ABB RAPID module: P101.mod

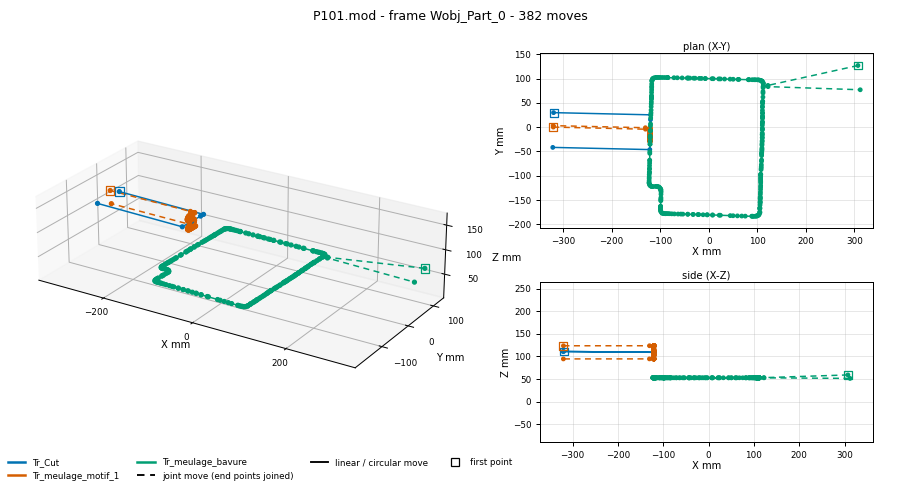
[picture p0: tool path of P101.mod in frame Wobj_Part_0, 382 of 390 moves have a stored position in this frame; points joined in program order, loops and branches not executed]
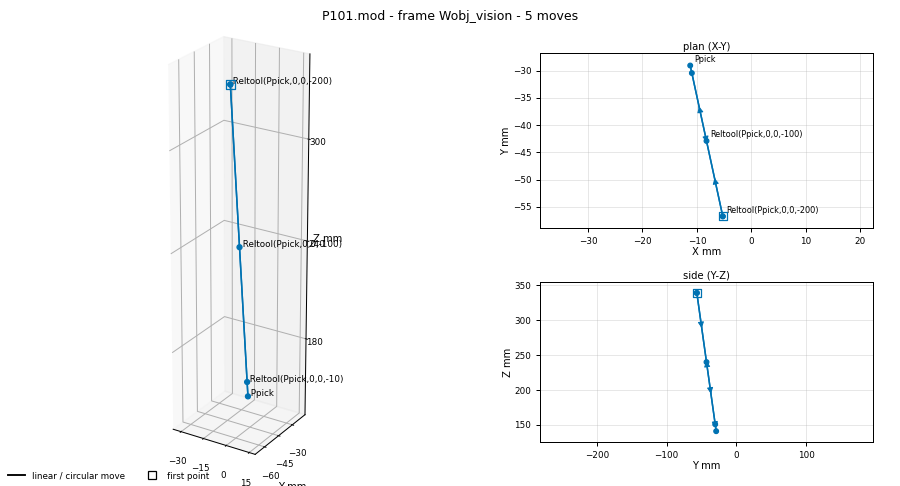
[picture p1: tool path of P101.mod in frame Wobj_vision, 5 of 390 moves have a stored position in this frame; points joined in program order, loops and branches not executed]
MODULE P101
	LOCAL CONST Speeddata vitesse_Tronconnage :=[10, 500, 0, 0];
	LOCAL CONST Robtarget Coupe_0 :=[[-120.682296875,-15.2756298828125,109.2198984375],[0.707017403537071,0.707090697782449,-0.00476918331892896,-0.01124237945003],[0,0,0,0],[8.999999E+09,8.999999E+09,8.999999E+09,8.999999E+09,8.999999E+09,8.999999E+09]];
	LOCAL CONST Robtarget Tr_meulage_motif_1_App1 :=[[-320.249128469475,0.246534065267081,123.638490401036],[0.494425938031671,-0.49422530691975,0.505508072978483,-0.505713284337244],[0,0,0,0],[8.999999E+09,8.999999E+09,8.999999E+09,8.999999E+09,8.999999E+09,8.999999E+09]];
	LOCAL CONST Robtarget Tr_meulage_motif_1_App2 :=[[-130.297538064099,-4.04151394615071,123.715605379427],[0.494425938031671,-0.49422530691975,0.505508072978483,-0.505713284337244],[0,0,0,0],[8.999999E+09,8.999999E+09,8.999999E+09,8.999999E+09,8.999999E+09,8.999999E+09]];
	LOCAL CONST Robtarget Tr_meulage_motif_1_P0 :=[[-120.3000859375,-4.26720068359375,123.7196640625],[0.494425938031671,-0.49422530691975,0.505508072978483,-0.505713284337244],[0,0,0,0],[8.999999E+09,8.999999E+09,8.999999E+09,8.999999E+09,8.999999E+09,8.999999E+09]];
	LOCAL CONST Robtarget Tr_meulage_motif_1_P1 :=[[-120.322734375,-5.2669443359375,123.719625],[0.494425938031671,-0.49422530691975,0.505508072978483,-0.505713284337244],[0,0,0,0],[8.999999E+09,8.999999E+09,8.999999E+09,8.999999E+09,8.999999E+09,8.999999E+09]];
	LOCAL CONST Robtarget Tr_meulage_motif_1_P2 :=[[-120.3453828125,-6.26668798828125,123.71959375],[0.494425938031671,-0.49422530691975,0.505508072978483,-0.505713284337244],[0,0,0,0],[8.999999E+09,8.999999E+09,8.999999E+09,8.999999E+09,8.999999E+09,8.999999E+09]];
	LOCAL CONST Robtarget Tr_meulage_motif_1_P3 :=[[-120.36803125,-7.26643115234375,123.7195625],[0.494425938031671,-0.49422530691975,0.505508072978483,-0.505713284337244],[0,0,0,0],[8.999999E+09,8.999999E+09,8.999999E+09,8.999999E+09,8.999999E+09,8.999999E+09]];
	LOCAL CONST Robtarget Tr_meulage_motif_1_P4 :=[[-120.3906796875,-8.2661748046875,123.7195234375],[0.494425938031671,-0.49422530691975,0.505508072978483,-0.505713284337244],[0,0,0,0],[8.999999E+09,8.999999E+09,8.999999E+09,8.999999E+09,8.999999E+09,8.999999E+09]];
	LOCAL CONST Robtarget Tr_meulage_motif_1_P5 :=[[-120.413328125,-9.26591796875,123.7194921875],[0.494425938031671,-0.49422530691975,0.505508072978483,-0.505713284337244],[0,0,0,0],[8.999999E+09,8.999999E+09,8.999999E+09,8.999999E+09,8.999999E+09,8.999999E+09]];
	LOCAL CONST Robtarget Tr_meulage_motif_1_P6 :=[[-120.4359765625,-10.265662109375,123.7194609375],[0.494425938031671,-0.49422530691975,0.505508072978483,-0.505713284337244],[0,0,0,0],[8.999999E+09,8.999999E+09,8.999999E+09,8.999999E+09,8.999999E+09,8.999999E+09]];
	LOCAL CONST Robtarget Tr_meulage_motif_1_P7 :=[[-120.458625,-11.2654052734375,123.719421875],[0.494425938031671,-0.49422530691975,0.505508072978483,-0.505713284337244],[0,0,0,0],[8.999999E+09,8.999999E+09,8.999999E+09,8.999999E+09,8.999999E+09,8.999999E+09]];
	LOCAL CONST Robtarget Tr_meulage_motif_1_P8 :=[[-120.481265625,-12.2651484375,123.719390625],[0.494425938031671,-0.49422530691975,0.505508072978483,-0.505713284337244],[0,0,0,0],[8.999999E+09,8.999999E+09,8.999999E+09,8.999999E+09,8.999999E+09,8.999999E+09]];
	LOCAL CONST Robtarget Tr_meulage_motif_1_P9 :=[[-120.5039140625,-13.264892578125,123.719359375],[0.494425938031671,-0.49422530691975,0.505508072978483,-0.505713284337244],[0,0,0,0],[8.999999E+09,8.999999E+09,8.999999E+09,8.999999E+09,8.999999E+09,8.999999E+09]];
	LOCAL CONST Robtarget Tr_meulage_motif_1_P10 :=[[-120.5265625,-14.2646357421875,123.719328125],[0.494425938031671,-0.49422530691975,0.505508072978483,-0.505713284337244],[0,0,0,0],[8.999999E+09,8.999999E+09,8.999999E+09,8.999999E+09,8.999999E+09,8.999999E+09]];
	LOCAL CONST Robtarget Tr_meulage_motif_1_P11 :=[[-120.5492109375,-15.26437890625,123.7192890625],[0.494425938031671,-0.49422530691975,0.505508072978483,-0.505713284337244],[0,0,0,0],[8.999999E+09,8.999999E+09,8.999999E+09,8.999999E+09,8.999999E+09,8.999999E+09]];
	LOCAL CONST Robtarget Tr_meulage_motif_1_P12 :=[[-120.571859375,-16.264123046875,123.7192578125],[0.494425938031671,-0.49422530691975,0.505508072978483,-0.505713284337244],[0,0,0,0],[8.999999E+09,8.999999E+09,8.999999E+09,8.999999E+09,8.999999E+09,8.999999E+09]];
	LOCAL CONST Robtarget Tr_meulage_motif_1_P13 :=[[-120.5945078125,-17.2638671875,123.7192265625],[0.494425938031671,-0.49422530691975,0.505508072978483,-0.505713284337244],[0,0,0,0],[8.999999E+09,8.999999E+09,8.999999E+09,8.999999E+09,8.999999E+09,8.999999E+09]];
	LOCAL CONST Robtarget Tr_meulage_motif_1_P14 :=[[-120.61715625,-18.263609375,123.7191875],[0.494425938031671,-0.49422530691975,0.505508072978483,-0.505713284337244],[0,0,0,0],[8.999999E+09,8.999999E+09,8.999999E+09,8.999999E+09,8.999999E+09,8.999999E+09]];
	LOCAL CONST Robtarget Tr_meulage_motif_1_P15 :=[[-120.6398046875,-19.263353515625,123.71915625],[0.494425938031671,-0.49422530691975,0.505508072978483,-0.505713284337244],[0,0,0,0],[8.999999E+09,8.999999E+09,8.999999E+09,8.999999E+09,8.999999E+09,8.999999E+09]];
	LOCAL CONST Robtarget Tr_meulage_motif_1_P16 :=[[-120.662453125,-20.26309765625,123.719125],[0.494425938031671,-0.49422530691975,0.505508072978483,-0.505713284337244],[0,0,0,0],[8.999999E+09,8.999999E+09,8.999999E+09,8.999999E+09,8.999999E+09,8.999999E+09]];
	LOCAL CONST Robtarget Tr_meulage_motif_1_P17 :=[[-120.6851015625,-21.26283984375,123.7190859375],[0.494425938031671,-0.49422530691975,0.505508072978483,-0.505713284337244],[0,0,0,0],[8.999999E+09,8.999999E+09,8.999999E+09,8.999999E+09,8.999999E+09,8.999999E+09]];
	LOCAL CONST Robtarget Tr_meulage_motif_1_P18 :=[[-120.70775,-22.262583984375,123.7190546875],[0.494425938031671,-0.49422530691975,0.505508072978483,-0.505713284337244],[0,0,0,0],[8.999999E+09,8.999999E+09,8.999999E+09,8.999999E+09,8.999999E+09,8.999999E+09]];
	LOCAL CONST Robtarget Tr_meulage_motif_1_P19 :=[[-120.7312421875,-23.254865234375,123.6084296875],[0.494425938031671,-0.49422530691975,0.505508072978483,-0.505713284337244],[0,0,0,0],[8.999999E+09,8.999999E+09,8.999999E+09,8.999999E+09,8.999999E+09,8.999999E+09]];
	LOCAL CONST Robtarget Tr_meulage_motif_1_P20 :=[[-120.754609375,-24.201072265625,123.39721875],[0.494425938031671,-0.49422530691975,0.505508072978483,-0.505713284337244],[0,0,0,0],[8.999999E+09,8.999999E+09,8.999999E+09,8.999999E+09,8.999999E+09,8.999999E+09]];
	LOCAL CONST Robtarget Tr_meulage_motif_1_P21 :=[[-120.7764140625,-25.053505859375,123.125359375],[0.494425938031671,-0.49422530691975,0.505508072978483,-0.505713284337244],[0,0,0,0],[8.999999E+09,8.999999E+09,8.999999E+09,8.999999E+09,8.999999E+09,8.999999E+09]];
	LOCAL CONST Robtarget Tr_meulage_motif_1_P22 :=[[-120.795921875,-25.80318359375,122.84940625],[0.494425938031671,-0.49422530691975,0.505508072978483,-0.505713284337244],[0,0,0,0],[8.999999E+09,8.999999E+09,8.999999E+09,8.999999E+09,8.999999E+09,8.999999E+09]];
	LOCAL CONST Robtarget Tr_meulage_motif_1_P23 :=[[-120.8265,-26.90381640625,122.2332734375],[0.494425938031671,-0.49422530691975,0.505508072978483,-0.505713284337244],[0,0,0,0],[8.999999E+09,8.999999E+09,8.999999E+09,8.999999E+09,8.999999E+09,8.999999E+09]];
	LOCAL CONST Robtarget Tr_meulage_motif_1_P24 :=[[-120.8574453125,-27.927224609375,121.3856171875],[0.494425938031671,-0.49422530691975,0.505508072978483,-0.505713284337244],[0,0,0,0],[8.999999E+09,8.999999E+09,8.999999E+09,8.999999E+09,8.999999E+09,8.999999E+09]];
	LOCAL CONST Robtarget Tr_meulage_motif_1_P25 :=[[-120.8860234375,-28.774416015625,120.3617578125],[0.494425938031671,-0.49422530691975,0.505508072978483,-0.505713284337244],[0,0,0,0],[8.999999E+09,8.999999E+09,8.999999E+09,8.999999E+09,8.999999E+09,8.999999E+09]];
	LOCAL CONST Robtarget Tr_meulage_motif_1_P26 :=[[-120.907296875,-29.262177734375,119.2456015625],[0.494425938031671,-0.49422530691975,0.505508072978483,-0.505713284337244],[0,0,0,0],[8.999999E+09,8.999999E+09,8.999999E+09,8.999999E+09,8.999999E+09,8.999999E+09]];
	LOCAL CONST Robtarget Tr_meulage_motif_1_P27 :=[[-120.91428125,-29.28906640625,118.5496640625],[0.494425938031671,-0.49422530691975,0.505508072978483,-0.505713284337244],[0,0,0,0],[8.999999E+09,8.999999E+09,8.999999E+09,8.999999E+09,8.999999E+09,8.999999E+09]];
	LOCAL CONST Robtarget Tr_meulage_motif_1_P28 :=[[-120.9203359375,-29.28890625,117.8884375],[0.494425938031671,-0.49422530691975,0.505508072978483,-0.505713284337244],[0,0,0,0],[8.999999E+09,8.999999E+09,8.999999E+09,8.999999E+09,8.999999E+09,8.999999E+09]];
	LOCAL CONST Robtarget Tr_meulage_motif_1_P29 :=[[-120.925140625,-29.23388671875,117.227375],[0.494425938031671,-0.49422530691975,0.505508072978483,-0.505713284337244],[0,0,0,0],[8.999999E+09,8.999999E+09,8.999999E+09,8.999999E+09,8.999999E+09,8.999999E+09]];
	LOCAL CONST Robtarget Tr_meulage_motif_1_P30 :=[[-120.9239453125,-28.735529296875,116.1256875],[0.494425938031671,-0.49422530691975,0.505508072978483,-0.505713284337244],[0,0,0,0],[8.999999E+09,8.999999E+09,8.999999E+09,8.999999E+09,8.999999E+09,8.999999E+09]];
	LOCAL CONST Robtarget Tr_meulage_motif_1_P31 :=[[-120.9137578125,-27.878880859375,115.1191328125],[0.494425938031671,-0.49422530691975,0.505508072978483,-0.505713284337244],[0,0,0,0],[8.999999E+09,8.999999E+09,8.999999E+09,8.999999E+09,8.999999E+09,8.999999E+09]];
	LOCAL CONST Robtarget Tr_meulage_motif_1_P32 :=[[-120.898171875,-26.855537109375,114.290328125],[0.494425938031671,-0.49422530691975,0.505508072978483,-0.505713284337244],[0,0,0,0],[8.999999E+09,8.999999E+09,8.999999E+09,8.999999E+09,8.999999E+09,8.999999E+09]];
	LOCAL CONST Robtarget Tr_meulage_motif_1_P33 :=[[-120.886234375,-26.168525390625,113.8946171875],[0.494425938031671,-0.49422530691975,0.505508072978483,-0.505713284337244],[0,0,0,0],[8.999999E+09,8.999999E+09,8.999999E+09,8.999999E+09,8.999999E+09,8.999999E+09]];
	LOCAL CONST Robtarget Tr_meulage_motif_1_P34 :=[[-120.86446875,-25.010548828125,113.4071484375],[0.494425938031671,-0.49422530691975,0.505508072978483,-0.505713284337244],[0,0,0,0],[8.999999E+09,8.999999E+09,8.999999E+09,8.999999E+09,8.999999E+09,8.999999E+09]];
	LOCAL CONST Robtarget Tr_meulage_motif_1_P35 :=[[-120.8477421875,-24.165669921875,113.14309375],[0.494425938031671,-0.49422530691975,0.505508072978483,-0.505713284337244],[0,0,0,0],[8.999999E+09,8.999999E+09,8.999999E+09,8.999999E+09,8.999999E+09,8.999999E+09]];
	LOCAL CONST Robtarget Tr_meulage_motif_1_P36 :=[[-120.8285078125,-23.233859375,112.9386640625],[0.494425938031671,-0.49422530691975,0.505508072978483,-0.505713284337244],[0,0,0,0],[8.999999E+09,8.999999E+09,8.999999E+09,8.999999E+09,8.999999E+09,8.999999E+09]];
	LOCAL CONST Robtarget Tr_meulage_motif_1_P37 :=[[-120.8072734375,-22.2525234375,112.830109375],[0.494425938031671,-0.49422530691975,0.505508072978483,-0.505713284337244],[0,0,0,0],[8.999999E+09,8.999999E+09,8.999999E+09,8.999999E+09,8.999999E+09,8.999999E+09]];
	LOCAL CONST Robtarget Tr_meulage_motif_1_P38 :=[[-120.7858046875,-21.2601875,112.719546875],[0.494425938031671,-0.49422530691975,0.505508072978483,-0.505713284337244],[0,0,0,0],[8.999999E+09,8.999999E+09,8.999999E+09,8.999999E+09,8.999999E+09,8.999999E+09]];
	LOCAL CONST Robtarget Tr_meulage_motif_1_P39 :=[[-120.76315625,-20.2604453125,112.7195859375],[0.494425938031671,-0.49422530691975,0.505508072978483,-0.505713284337244],[0,0,0,0],[8.999999E+09,8.999999E+09,8.999999E+09,8.999999E+09,8.999999E+09,8.999999E+09]];
	LOCAL CONST Robtarget Tr_meulage_motif_1_P40 :=[[-120.7405078125,-19.260701171875,112.7196171875],[0.494425938031671,-0.49422530691975,0.505508072978483,-0.505713284337244],[0,0,0,0],[8.999999E+09,8.999999E+09,8.999999E+09,8.999999E+09,8.999999E+09,8.999999E+09]];
	LOCAL CONST Robtarget Tr_meulage_motif_1_P41 :=[[-120.7178671875,-18.26095703125,112.7196484375],[0.494425938031671,-0.49422530691975,0.505508072978483,-0.505713284337244],[0,0,0,0],[8.999999E+09,8.999999E+09,8.999999E+09,8.999999E+09,8.999999E+09,8.999999E+09]];
	LOCAL CONST Robtarget Tr_meulage_motif_1_P42 :=[[-120.69521875,-17.26121484375,112.7196875],[0.494425938031671,-0.49422530691975,0.505508072978483,-0.505713284337244],[0,0,0,0],[8.999999E+09,8.999999E+09,8.999999E+09,8.999999E+09,8.999999E+09,8.999999E+09]];
	LOCAL CONST Robtarget Tr_meulage_motif_1_P43 :=[[-120.6725703125,-16.261470703125,112.71971875],[0.494425938031671,-0.49422530691975,0.505508072978483,-0.505713284337244],[0,0,0,0],[8.999999E+09,8.999999E+09,8.999999E+09,8.999999E+09,8.999999E+09,8.999999E+09]];
	LOCAL CONST Robtarget Tr_meulage_motif_1_P44 :=[[-120.649921875,-15.2617275390625,112.71975],[0.494425938031671,-0.49422530691975,0.505508072978483,-0.505713284337244],[0,0,0,0],[8.999999E+09,8.999999E+09,8.999999E+09,8.999999E+09,8.999999E+09,8.999999E+09]];
	LOCAL CONST Robtarget Tr_meulage_motif_1_P45 :=[[-120.6272734375,-14.261984375,112.7197890625],[0.494425938031671,-0.49422530691975,0.505508072978483,-0.505713284337244],[0,0,0,0],[8.999999E+09,8.999999E+09,8.999999E+09,8.999999E+09,8.999999E+09,8.999999E+09]];
	LOCAL CONST Robtarget Tr_meulage_motif_1_P46 :=[[-120.604625,-13.262240234375,112.7198203125],[0.494425938031671,-0.49422530691975,0.505508072978483,-0.505713284337244],[0,0,0,0],[8.999999E+09,8.999999E+09,8.999999E+09,8.999999E+09,8.999999E+09,8.999999E+09]];
	LOCAL CONST Robtarget Tr_meulage_motif_1_P47 :=[[-120.5819765625,-12.2624970703125,112.7198515625],[0.494425938031671,-0.49422530691975,0.505508072978483,-0.505713284337244],[0,0,0,0],[8.999999E+09,8.999999E+09,8.999999E+09,8.999999E+09,8.999999E+09,8.999999E+09]];
	LOCAL CONST Robtarget Tr_meulage_motif_1_P48 :=[[-120.559328125,-11.26275390625,112.719890625],[0.494425938031671,-0.49422530691975,0.505508072978483,-0.505713284337244],[0,0,0,0],[8.999999E+09,8.999999E+09,8.999999E+09,8.999999E+09,8.999999E+09,8.999999E+09]];
	LOCAL CONST Robtarget Tr_meulage_motif_1_P49 :=[[-120.537859375,-10.2704189453125,112.609328125],[0.494425938031671,-0.49422530691975,0.505508072978483,-0.505713284337244],[0,0,0,0],[8.999999E+09,8.999999E+09,8.999999E+09,8.999999E+09,8.999999E+09,8.999999E+09]];
	LOCAL CONST Robtarget Tr_meulage_motif_1_P50 :=[[-120.518359375,-9.3241103515625,112.3981875],[0.494425938031671,-0.49422530691975,0.505508072978483,-0.505713284337244],[0,0,0,0],[8.999999E+09,8.999999E+09,8.999999E+09,8.999999E+09,8.999999E+09,8.999999E+09]];
	LOCAL CONST Robtarget Tr_meulage_motif_1_P51 :=[[-120.50153125,-8.471544921875,112.1263828125],[0.494425938031671,-0.49422530691975,0.505508072978483,-0.505713284337244],[0,0,0,0],[8.999999E+09,8.999999E+09,8.999999E+09,8.999999E+09,8.999999E+09,8.999999E+09]];
	LOCAL CONST Robtarget Tr_meulage_motif_1_P52 :=[[-120.488203125,-7.760154296875,111.8222578125],[0.494425938031671,-0.49422530691975,0.505508072978483,-0.505713284337244],[0,0,0,0],[8.999999E+09,8.999999E+09,8.999999E+09,8.999999E+09,8.999999E+09,8.999999E+09]];
	LOCAL CONST Robtarget Tr_meulage_motif_1_P53 :=[[-120.47084375,-6.725791015625,111.1597890625],[0.494425938031671,-0.49422530691975,0.505508072978483,-0.505713284337244],[0,0,0,0],[8.999999E+09,8.999999E+09,8.999999E+09,8.999999E+09,8.999999E+09,8.999999E+09]];
	LOCAL CONST Robtarget Tr_meulage_motif_1_P54 :=[[-120.458671875,-5.82386767578125,110.257921875],[0.494425938031671,-0.49422530691975,0.505508072978483,-0.505713284337244],[0,0,0,0],[8.999999E+09,8.999999E+09,8.999999E+09,8.999999E+09,8.999999E+09,8.999999E+09]];
	LOCAL CONST Robtarget Tr_meulage_motif_1_P55 :=[[-120.4561328125,-5.28878369140625,109.211953125],[0.494425938031671,-0.49422530691975,0.505508072978483,-0.505713284337244],[0,0,0,0],[8.999999E+09,8.999999E+09,8.999999E+09,8.999999E+09,8.999999E+09,8.999999E+09]];
	LOCAL CONST Robtarget Tr_meulage_motif_1_P56 :=[[-120.458296875,-5.1038828125,108.5187734375],[0.494425938031671,-0.49422530691975,0.505508072978483,-0.505713284337244],[0,0,0,0],[8.999999E+09,8.999999E+09,8.999999E+09,8.999999E+09,8.999999E+09,8.999999E+09]];
	LOCAL CONST Robtarget Tr_meulage_motif_1_P57 :=[[-120.4638984375,-5.0398701171875,107.7488046875],[0.494425938031671,-0.49422530691975,0.505508072978483,-0.505713284337244],[0,0,0,0],[8.999999E+09,8.999999E+09,8.999999E+09,8.999999E+09,8.999999E+09,8.999999E+09]];
	LOCAL CONST Robtarget Tr_meulage_motif_1_P58 :=[[-120.4724609375,-5.1066044921875,106.9789609375],[0.494425938031671,-0.49422530691975,0.505508072978483,-0.505713284337244],[0,0,0,0],[8.999999E+09,8.999999E+09,8.999999E+09,8.999999E+09,8.999999E+09,8.999999E+09]];
	LOCAL CONST Robtarget Tr_meulage_motif_1_P59 :=[[-120.492109375,-5.52582373046875,105.8707421875],[0.494425938031671,-0.49422530691975,0.505508072978483,-0.505713284337244],[0,0,0,0],[8.999999E+09,8.999999E+09,8.999999E+09,8.999999E+09,8.999999E+09,8.999999E+09]];
	LOCAL CONST Robtarget Tr_meulage_motif_1_P60 :=[[-120.506859375,-5.939888671875,105.2850625],[0.494425938031671,-0.49422530691975,0.505508072978483,-0.505713284337244],[0,0,0,0],[8.999999E+09,8.999999E+09,8.999999E+09,8.999999E+09,8.999999E+09,8.999999E+09]];
	LOCAL CONST Robtarget Tr_meulage_motif_1_P61 :=[[-120.5350703125,-6.826572265625,104.3979453125],[0.494425938031671,-0.49422530691975,0.505508072978483,-0.505713284337244],[0,0,0,0],[8.999999E+09,8.999999E+09,8.999999E+09,8.999999E+09,8.999999E+09,8.999999E+09]];
	LOCAL CONST Robtarget Tr_meulage_motif_1_P62 :=[[-120.552125,-7.412009765625,103.9836328125],[0.494425938031671,-0.49422530691975,0.505508072978483,-0.505713284337244],[0,0,0,0],[8.999999E+09,8.999999E+09,8.999999E+09,8.999999E+09,8.999999E+09,8.999999E+09]];
	LOCAL CONST Robtarget Tr_meulage_motif_1_P63 :=[[-120.5824296875,-8.529498046875,103.4395234375],[0.494425938031671,-0.49422530691975,0.505508072978483,-0.505713284337244],[0,0,0,0],[8.999999E+09,8.999999E+09,8.999999E+09,8.999999E+09,8.999999E+09,8.999999E+09]];
	LOCAL CONST Robtarget Tr_meulage_motif_1_P64 :=[[-120.603828125,-9.35480859375,103.1440078125],[0.494425938031671,-0.49422530691975,0.505508072978483,-0.505713284337244],[0,0,0,0],[8.999999E+09,8.999999E+09,8.999999E+09,8.999999E+09,8.999999E+09,8.999999E+09]];
	LOCAL CONST Robtarget Tr_meulage_motif_1_P65 :=[[-120.6268125,-10.2865205078125,102.939515625],[0.494425938031671,-0.49422530691975,0.505508072978483,-0.505713284337244],[0,0,0,0],[8.999999E+09,8.999999E+09,8.999999E+09,8.999999E+09,8.999999E+09,8.999999E+09]];
	LOCAL CONST Robtarget Tr_meulage_motif_1_P66 :=[[-120.6500390625,-11.2678046875,102.8308984375],[0.494425938031671,-0.49422530691975,0.505508072978483,-0.505713284337244],[0,0,0,0],[8.999999E+09,8.999999E+09,8.999999E+09,8.999999E+09,8.999999E+09,8.999999E+09]];
	LOCAL CONST Robtarget Tr_meulage_motif_1_P67 :=[[-120.67353125,-12.2600859375,102.7202734375],[0.494425938031671,-0.49422530691975,0.505508072978483,-0.505713284337244],[0,0,0,0],[8.999999E+09,8.999999E+09,8.999999E+09,8.999999E+09,8.999999E+09,8.999999E+09]];
	LOCAL CONST Robtarget Tr_meulage_motif_1_P68 :=[[-120.696171875,-13.259830078125,102.7202421875],[0.494425938031671,-0.49422530691975,0.505508072978483,-0.505713284337244],[0,0,0,0],[8.999999E+09,8.999999E+09,8.999999E+09,8.999999E+09,8.999999E+09,8.999999E+09]];
	LOCAL CONST Robtarget Tr_meulage_motif_1_P69 :=[[-120.7188203125,-14.2595732421875,102.720203125],[0.494425938031671,-0.49422530691975,0.505508072978483,-0.505713284337244],[0,0,0,0],[8.999999E+09,8.999999E+09,8.999999E+09,8.999999E+09,8.999999E+09,8.999999E+09]];
	LOCAL CONST Robtarget Tr_meulage_motif_1_P70 :=[[-120.74146875,-15.25931640625,102.720171875],[0.494425938031671,-0.49422530691975,0.505508072978483,-0.505713284337244],[0,0,0,0],[8.999999E+09,8.999999E+09,8.999999E+09,8.999999E+09,8.999999E+09,8.999999E+09]];
	LOCAL CONST Robtarget Tr_meulage_motif_1_P71 :=[[-120.7641171875,-16.259060546875,102.720140625],[0.494425938031671,-0.49422530691975,0.505508072978483,-0.505713284337244],[0,0,0,0],[8.999999E+09,8.999999E+09,8.999999E+09,8.999999E+09,8.999999E+09,8.999999E+09]];
	LOCAL CONST Robtarget Tr_meulage_motif_1_P72 :=[[-120.786765625,-17.258802734375,102.7201015625],[0.494425938031671,-0.49422530691975,0.505508072978483,-0.505713284337244],[0,0,0,0],[8.999999E+09,8.999999E+09,8.999999E+09,8.999999E+09,8.999999E+09,8.999999E+09]];
	LOCAL CONST Robtarget Tr_meulage_motif_1_P73 :=[[-120.8094140625,-18.258546875,102.7200703125],[0.494425938031671,-0.49422530691975,0.505508072978483,-0.505713284337244],[0,0,0,0],[8.999999E+09,8.999999E+09,8.999999E+09,8.999999E+09,8.999999E+09,8.999999E+09]];
	LOCAL CONST Robtarget Tr_meulage_motif_1_P74 :=[[-120.8320625,-19.258291015625,102.7200390625],[0.494425938031671,-0.49422530691975,0.505508072978483,-0.505713284337244],[0,0,0,0],[8.999999E+09,8.999999E+09,8.999999E+09,8.999999E+09,8.999999E+09,8.999999E+09]];
	LOCAL CONST Robtarget Tr_meulage_motif_1_P75 :=[[-120.8547109375,-20.258033203125,102.72],[0.494425938031671,-0.49422530691975,0.505508072978483,-0.505713284337244],[0,0,0,0],[8.999999E+09,8.999999E+09,8.999999E+09,8.999999E+09,8.999999E+09,8.999999E+09]];
	LOCAL CONST Robtarget Tr_meulage_motif_1_P76 :=[[-120.877359375,-21.25777734375,102.71996875],[0.494425938031671,-0.49422530691975,0.505508072978483,-0.505713284337244],[0,0,0,0],[8.999999E+09,8.999999E+09,8.999999E+09,8.999999E+09,8.999999E+09,8.999999E+09]];
	LOCAL CONST Robtarget Tr_meulage_motif_1_P77 :=[[-120.9000078125,-22.257521484375,102.7199375],[0.494425938031671,-0.49422530691975,0.505508072978483,-0.505713284337244],[0,0,0,0],[8.999999E+09,8.999999E+09,8.999999E+09,8.999999E+09,8.999999E+09,8.999999E+09]];
	LOCAL CONST Robtarget Tr_meulage_motif_1_P78 :=[[-120.9235,-23.249802734375,102.6093125],[0.494425938031671,-0.49422530691975,0.505508072978483,-0.505713284337244],[0,0,0,0],[8.999999E+09,8.999999E+09,8.999999E+09,8.999999E+09,8.999999E+09,8.999999E+09]];
	LOCAL CONST Robtarget Tr_meulage_motif_1_P79 :=[[-120.9468671875,-24.1960078125,102.3981015625],[0.494425938031671,-0.49422530691975,0.505508072978483,-0.505713284337244],[0,0,0,0],[8.999999E+09,8.999999E+09,8.999999E+09,8.999999E+09,8.999999E+09,8.999999E+09]];
	LOCAL CONST Robtarget Tr_meulage_motif_1_P80 :=[[-120.968671875,-25.048443359375,102.1262421875],[0.494425938031671,-0.49422530691975,0.505508072978483,-0.505713284337244],[0,0,0,0],[8.999999E+09,8.999999E+09,8.999999E+09,8.999999E+09,8.999999E+09,8.999999E+09]];
	LOCAL CONST Robtarget Tr_meulage_motif_1_P81 :=[[-120.9881796875,-25.79812109375,101.8502890625],[0.494425938031671,-0.49422530691975,0.505508072978483,-0.505713284337244],[0,0,0,0],[8.999999E+09,8.999999E+09,8.999999E+09,8.999999E+09,8.999999E+09,8.999999E+09]];
	LOCAL CONST Robtarget Tr_meulage_motif_1_P82 :=[[-121.0187578125,-26.89875390625,101.23415625],[0.494425938031671,-0.49422530691975,0.505508072978483,-0.505713284337244],[0,0,0,0],[8.999999E+09,8.999999E+09,8.999999E+09,8.999999E+09,8.999999E+09,8.999999E+09]];
	LOCAL CONST Robtarget Tr_meulage_motif_1_P83 :=[[-121.048609375,-27.85501171875,100.3401875],[0.494425938031671,-0.49422530691975,0.505508072978483,-0.505713284337244],[0,0,0,0],[8.999999E+09,8.999999E+09,8.999999E+09,8.999999E+09,8.999999E+09,8.999999E+09]];
	LOCAL CONST Robtarget Tr_meulage_motif_1_P84 :=[[-121.07234375,-28.46371875,99.25421875],[0.494425938031671,-0.49422530691975,0.505508072978483,-0.505713284337244],[0,0,0,0],[8.999999E+09,8.999999E+09,8.999999E+09,8.999999E+09,8.999999E+09,8.999999E+09]];
	LOCAL CONST Robtarget Tr_meulage_motif_1_P85 :=[[-121.0851953125,-28.63275,98.269875],[0.494425938031671,-0.49422530691975,0.505508072978483,-0.505713284337244],[0,0,0,0],[8.999999E+09,8.999999E+09,8.999999E+09,8.999999E+09,8.999999E+09,8.999999E+09]];
	LOCAL CONST Robtarget Tr_meulage_motif_1_P86 :=[[-121.08409375,-28.501265625,98.065234375],[0.494425938031671,-0.49422530691975,0.505508072978483,-0.505713284337244],[0,0,0,0],[8.999999E+09,8.999999E+09,8.999999E+09,8.999999E+09,8.999999E+09,8.999999E+09]];
	LOCAL CONST Robtarget Tr_meulage_motif_1_P87 :=[[-121.0879453125,-28.377748046875,97.338859375],[0.494425938031671,-0.49422530691975,0.505508072978483,-0.505713284337244],[0,0,0,0],[8.999999E+09,8.999999E+09,8.999999E+09,8.999999E+09,8.999999E+09,8.999999E+09]];
	LOCAL CONST Robtarget Tr_meulage_motif_1_P88 :=[[-121.08103125,-27.693697265625,96.402015625],[0.494425938031671,-0.49422530691975,0.505508072978483,-0.505713284337244],[0,0,0,0],[8.999999E+09,8.999999E+09,8.999999E+09,8.999999E+09,8.999999E+09,8.999999E+09]];
	LOCAL CONST Robtarget Tr_meulage_motif_1_P89 :=[[-121.0726484375,-27.136103515625,95.9382421875],[0.494425938031671,-0.49422530691975,0.505508072978483,-0.505713284337244],[0,0,0,0],[8.999999E+09,8.999999E+09,8.999999E+09,8.999999E+09,8.999999E+09,8.999999E+09]];
	LOCAL CONST Robtarget Tr_meulage_motif_1_P90 :=[[-121.05190625,-26.005953125,95.4078671875],[0.494425938031671,-0.49422530691975,0.505508072978483,-0.505713284337244],[0,0,0,0],[8.999999E+09,8.999999E+09,8.999999E+09,8.999999E+09,8.999999E+09,8.999999E+09]];
	LOCAL CONST Robtarget Tr_meulage_motif_1_P91 :=[[-121.0351875,-25.16107421875,95.1438125],[0.494425938031671,-0.49422530691975,0.505508072978483,-0.505713284337244],[0,0,0,0],[8.999999E+09,8.999999E+09,8.999999E+09,8.999999E+09,8.999999E+09,8.999999E+09]];
	LOCAL CONST Robtarget Tr_meulage_motif_1_P92 :=[[-121.015953125,-24.229263671875,94.9393828125],[0.494425938031671,-0.49422530691975,0.505508072978483,-0.505713284337244],[0,0,0,0],[8.999999E+09,8.999999E+09,8.999999E+09,8.999999E+09,8.999999E+09,8.999999E+09]];
	LOCAL CONST Robtarget Tr_meulage_motif_1_P93 :=[[-120.99471875,-23.247927734375,94.830828125],[0.494425938031671,-0.49422530691975,0.505508072978483,-0.505713284337244],[0,0,0,0],[8.999999E+09,8.999999E+09,8.999999E+09,8.999999E+09,8.999999E+09,8.999999E+09]];
	LOCAL CONST Robtarget Tr_meulage_motif_1_P94 :=[[-120.97325,-22.255591796875,94.7202734375],[0.494425938031671,-0.49422530691975,0.505508072978483,-0.505713284337244],[0,0,0,0],[8.999999E+09,8.999999E+09,8.999999E+09,8.999999E+09,8.999999E+09,8.999999E+09]];
	LOCAL CONST Robtarget Tr_meulage_motif_1_P95 :=[[-120.9506015625,-21.255849609375,94.7203046875],[0.494425938031671,-0.49422530691975,0.505508072978483,-0.505713284337244],[0,0,0,0],[8.999999E+09,8.999999E+09,8.999999E+09,8.999999E+09,8.999999E+09,8.999999E+09]];
	LOCAL CONST Robtarget Tr_meulage_motif_1_P96 :=[[-120.927953125,-20.25610546875,94.7203359375],[0.494425938031671,-0.49422530691975,0.505508072978483,-0.505713284337244],[0,0,0,0],[8.999999E+09,8.999999E+09,8.999999E+09,8.999999E+09,8.999999E+09,8.999999E+09]];
	LOCAL CONST Robtarget Tr_meulage_motif_1_P97 :=[[-120.9053046875,-19.256361328125,94.720375],[0.494425938031671,-0.49422530691975,0.505508072978483,-0.505713284337244],[0,0,0,0],[8.999999E+09,8.999999E+09,8.999999E+09,8.999999E+09,8.999999E+09,8.999999E+09]];
	LOCAL CONST Robtarget Tr_meulage_motif_1_P98 :=[[-120.88265625,-18.256619140625,94.72040625],[0.494425938031671,-0.49422530691975,0.505508072978483,-0.505713284337244],[0,0,0,0],[8.999999E+09,8.999999E+09,8.999999E+09,8.999999E+09,8.999999E+09,8.999999E+09]];
	LOCAL CONST Robtarget Tr_meulage_motif_1_P99 :=[[-120.8600078125,-17.256875,94.7204375],[0.494425938031671,-0.49422530691975,0.505508072978483,-0.505713284337244],[0,0,0,0],[8.999999E+09,8.999999E+09,8.999999E+09,8.999999E+09,8.999999E+09,8.999999E+09]];
	LOCAL CONST Robtarget Tr_meulage_motif_1_P100 :=[[-120.837359375,-16.2571318359375,94.7204765625],[0.494425938031671,-0.49422530691975,0.505508072978483,-0.505713284337244],[0,0,0,0],[8.999999E+09,8.999999E+09,8.999999E+09,8.999999E+09,8.999999E+09,8.999999E+09]];
	LOCAL CONST Robtarget Tr_meulage_motif_1_P101 :=[[-120.8147109375,-15.2573876953125,94.7205078125],[0.494425938031671,-0.49422530691975,0.505508072978483,-0.505713284337244],[0,0,0,0],[8.999999E+09,8.999999E+09,8.999999E+09,8.999999E+09,8.999999E+09,8.999999E+09]];
	LOCAL CONST Robtarget Tr_meulage_motif_1_P102 :=[[-120.7920625,-14.25764453125,94.7205390625],[0.494425938031671,-0.49422530691975,0.505508072978483,-0.505713284337244],[0,0,0,0],[8.999999E+09,8.999999E+09,8.999999E+09,8.999999E+09,8.999999E+09,8.999999E+09]];
	LOCAL CONST Robtarget Tr_meulage_motif_1_P103 :=[[-120.7694140625,-13.2579013671875,94.720578125],[0.494425938031671,-0.49422530691975,0.505508072978483,-0.505713284337244],[0,0,0,0],[8.999999E+09,8.999999E+09,8.999999E+09,8.999999E+09,8.999999E+09,8.999999E+09]];
	LOCAL CONST Robtarget Tr_meulage_motif_1_P104 :=[[-120.746765625,-12.2581572265625,94.720609375],[0.494425938031671,-0.49422530691975,0.505508072978483,-0.505713284337244],[0,0,0,0],[8.999999E+09,8.999999E+09,8.999999E+09,8.999999E+09,8.999999E+09,8.999999E+09]];
	LOCAL CONST Robtarget Tr_meulage_motif_1_P105 :=[[-120.724125,-11.2584140625,94.720640625],[0.494425938031671,-0.49422530691975,0.505508072978483,-0.505713284337244],[0,0,0,0],[8.999999E+09,8.999999E+09,8.999999E+09,8.999999E+09,8.999999E+09,8.999999E+09]];
	LOCAL CONST Robtarget Tr_meulage_motif_1_P106 :=[[-120.7014765625,-10.2586708984375,94.720671875],[0.494425938031671,-0.49422530691975,0.505508072978483,-0.505713284337244],[0,0,0,0],[8.999999E+09,8.999999E+09,8.999999E+09,8.999999E+09,8.999999E+09,8.999999E+09]];
	LOCAL CONST Robtarget Tr_meulage_motif_1_P107 :=[[-120.678828125,-9.2589267578125,94.7207109375],[0.494425938031671,-0.49422530691975,0.505508072978483,-0.505713284337244],[0,0,0,0],[8.999999E+09,8.999999E+09,8.999999E+09,8.999999E+09,8.999999E+09,8.999999E+09]];
	LOCAL CONST Robtarget Tr_meulage_motif_1_P108 :=[[-120.6561796875,-8.25918359375,94.7207421875],[0.494425938031671,-0.49422530691975,0.505508072978483,-0.505713284337244],[0,0,0,0],[8.999999E+09,8.999999E+09,8.999999E+09,8.999999E+09,8.999999E+09,8.999999E+09]];
	LOCAL CONST Robtarget Tr_meulage_motif_1_P109 :=[[-120.63353125,-7.25943994140625,94.7207734375],[0.494425938031671,-0.49422530691975,0.505508072978483,-0.505713284337244],[0,0,0,0],[8.999999E+09,8.999999E+09,8.999999E+09,8.999999E+09,8.999999E+09,8.999999E+09]];
	LOCAL CONST Robtarget Tr_meulage_motif_1_P110 :=[[-120.6108828125,-6.2596962890625,94.7208125],[0.494425938031671,-0.49422530691975,0.505508072978483,-0.505713284337244],[0,0,0,0],[8.999999E+09,8.999999E+09,8.999999E+09,8.999999E+09,8.999999E+09,8.999999E+09]];
	LOCAL CONST Robtarget Tr_meulage_motif_1_P111 :=[[-120.588234375,-5.259953125,94.72084375],[0.494425938031671,-0.49422530691975,0.505508072978483,-0.505713284337244],[0,0,0,0],[8.999999E+09,8.999999E+09,8.999999E+09,8.999999E+09,8.999999E+09,8.999999E+09]];
	LOCAL CONST Robtarget Tr_meulage_motif_1_P112 :=[[-120.5655859375,-4.26020947265625,94.720875],[0.494425938031671,-0.49422530691975,0.505508072978483,-0.505713284337244],[0,0,0,0],[8.999999E+09,8.999999E+09,8.999999E+09,8.999999E+09,8.999999E+09,8.999999E+09]];
	LOCAL CONST Robtarget Tr_meulage_motif_1_P113 :=[[-120.5429375,-3.26046606445313,94.7209140625],[0.494425938031671,-0.49422530691975,0.505508072978483,-0.505713284337244],[0,0,0,0],[8.999999E+09,8.999999E+09,8.999999E+09,8.999999E+09,8.999999E+09,8.999999E+09]];
	LOCAL CONST Robtarget Tr_meulage_motif_1_P114 :=[[-120.5202890625,-2.26072241210937,94.7209453125],[0.494425938031671,-0.49422530691975,0.505508072978483,-0.505713284337244],[0,0,0,0],[8.999999E+09,8.999999E+09,8.999999E+09,8.999999E+09,8.999999E+09,8.999999E+09]];
	LOCAL CONST Robtarget Tr_meulage_motif_1_P115 :=[[-120.497640625,-1.26097900390625,94.7209765625],[0.494425938031671,-0.49422530691975,0.505508072978483,-0.505713284337244],[0,0,0,0],[8.999999E+09,8.999999E+09,8.999999E+09,8.999999E+09,8.999999E+09,8.999999E+09]];
	LOCAL CONST Robtarget Tr_meulage_motif_1_degg1 :=[[-130.495092751599,-1.03529226646321,94.7169178794268],[0.494425938031671,-0.49422530691975,0.505508072978483,-0.505713284337244],[0,0,0,0],[8.999999E+09,8.999999E+09,8.999999E+09,8.999999E+09,8.999999E+09,8.999999E+09]];
	LOCAL CONST Robtarget Tr_meulage_motif_1_degg2 :=[[-320.446683156975,3.25275574495458,94.6398029010359],[0.494425938031671,-0.49422530691975,0.505508072978483,-0.505713284337244],[0,0,0,0],[8.999999E+09,8.999999E+09,8.999999E+09,8.999999E+09,8.999999E+09,8.999999E+09]];
	LOCAL CONST Robtarget Tr_meulage_bavure_App1 :=[[307.490240169758,127.130814114284,59.3046949992104],[0.435760329978366,-0.449720515650731,-0.559922490440299,0.542541424519013],[0,0,0,0],[8.999999E+09,8.999999E+09,8.999999E+09,8.999999E+09,8.999999E+09,8.999999E+09]];
	LOCAL CONST Robtarget Tr_meulage_bavure_App2 :=[[122.056313180363,86.1627157057142,53.3152347499605],[0.435760329978366,-0.449720515650731,-0.559922490440299,0.542541424519013],[0,0,0,0],[8.999999E+09,8.999999E+09,8.999999E+09,8.999999E+09,8.999999E+09,8.999999E+09]];
	LOCAL CONST Robtarget Tr_meulage_bavure_P0 :=[[112.2966328125,84.0065,53],[0.435760329978366,-0.449720515650731,-0.559922490440299,0.542541424519013],[0,0,0,0],[8.999999E+09,8.999999E+09,8.999999E+09,8.999999E+09,8.999999E+09,8.999999E+09]];
	LOCAL CONST Robtarget Tr_meulage_bavure_P1 :=[[112.45971875,89.4585546875,53],[0.4297745340756,-0.443501281000288,-0.56481980788287,0.54733814798017],[0,0,0,0],[8.999999E+09,8.999999E+09,8.999999E+09,8.999999E+09,8.999999E+09,8.999999E+09]];
	LOCAL CONST Robtarget Tr_meulage_bavure_P2 :=[[112.410765625,90.19153125,53],[0.411956238842138,-0.425004359099217,-0.57875503675503,0.560986594720753],[0,0,0,0],[8.999999E+09,8.999999E+09,8.999999E+09,8.999999E+09,8.999999E+09,8.999999E+09]];
	LOCAL CONST Robtarget Tr_meulage_bavure_P3 :=[[111.96734375,91.852046875,53],[0.382926483603339,-0.394892648932127,-0.599533491417809,0.581366232802458],[0,0,0,0],[8.999999E+09,8.999999E+09,8.999999E+09,8.999999E+09,8.999999E+09,8.999999E+09]];
	LOCAL CONST Robtarget Tr_meulage_bavure_P4 :=[[110.195890625,94.559390625,53],[0.344028718434338,-0.354582800936211,-0.623999051868104,0.605425851314895],[0,0,0,0],[8.999999E+09,8.999999E+09,8.999999E+09,8.999999E+09,8.999999E+09,8.999999E+09]];
	LOCAL CONST Robtarget Tr_meulage_bavure_P5 :=[[109.938234375,94.85275,53],[0.297547743603108,-0.306475395231743,-0.648729464342112,0.629831925587011],[0,0,0,0],[8.999999E+09,8.999999E+09,8.999999E+09,8.999999E+09,8.999999E+09,8.999999E+09]];
	LOCAL CONST Robtarget Tr_meulage_bavure_P6 :=[[109.3061796875,95.3077109375,53],[0.246841861880402,-0.254063270333085,-0.670720193319004,0.651655869432012],[0,0,0,0],[8.999999E+09,8.999999E+09,8.999999E+09,8.999999E+09,8.999999E+09,8.999999E+09]];
	LOCAL CONST Robtarget Tr_meulage_bavure_P7 :=[[107.198,96.4626484375,53],[0.196111566273891,-0.201695965554516,-0.68800720505713,0.668958202612173],[0,0,0,0],[8.999999E+09,8.999999E+09,8.999999E+09,8.999999E+09,8.999999E+09,8.999999E+09]];
	LOCAL CONST Robtarget Tr_meulage_bavure_P8 :=[[106.3204921875,96.67334375,53],[0.149408017681295,-0.153545625440822,-0.700056250966405,0.681191772295728],[0,0,0,0],[8.999999E+09,8.999999E+09,8.999999E+09,8.999999E+09,8.999999E+09,8.999999E+09]];
	LOCAL CONST Robtarget Tr_meulage_bavure_P9 :=[[102.95190625,97.5603671875,53],[0.109481885954018,-0.112431510203254,-0.707565253944476,0.689002382849186],[0,0,0,0],[8.999999E+09,8.999999E+09,8.999999E+09,8.999999E+09,8.999999E+09,8.999999E+09]];
	LOCAL CONST Robtarget Tr_meulage_bavure_P10 :=[[100.802828125,97.68603125,53],[0.0773783631448703,-0.0794099398417434,-0.711793043631003,0.69358295351736],[0,0,0,0],[8.999999E+09,8.999999E+09,8.999999E+09,8.999999E+09,8.999999E+09,8.999999E+09]];
	LOCAL CONST Robtarget Tr_meulage_bavure_P11 :=[[96.409546875,97.845578125,53],[0.052876417674232,-0.0542321705616713,-0.713942985192362,0.696095086913224],[0,0,0,0],[8.999999E+09,8.999999E+09,8.999999E+09,8.999999E+09,8.999999E+09,8.999999E+09]];
	LOCAL CONST Robtarget Tr_meulage_bavure_P12 :=[[93.62884375,97.83578125,53],[0.035062643335608,-0.0359434286222219,-0.714919944705722,0.697400999169894],[0,0,0,0],[8.999999E+09,8.999999E+09,8.999999E+09,8.999999E+09,8.999999E+09,8.999999E+09]];
	LOCAL CONST Robtarget Tr_meulage_bavure_P13 :=[[89.628265625,97.90740625,53],[0.0228122292977511,-0.0233757666492771,-0.715299032469505,0.698054775699024],[0,0,0,0],[8.999999E+09,8.999999E+09,8.999999E+09,8.999999E+09,8.999999E+09,8.999999E+09]];
	LOCAL CONST Robtarget Tr_meulage_bavure_P14 :=[[83.3127109375,97.9175703125,53],[0.0149825157169001,-0.0153477690350964,-0.715405638983986,0.698380084136392],[0,0,0,0],[8.999999E+09,8.999999E+09,8.999999E+09,8.999999E+09,8.999999E+09,8.999999E+09]];
	LOCAL CONST Robtarget Tr_meulage_bavure_P15 :=[[82.4075625,97.918609375,53],[0.010484872452233,-0.0107379672553927,-0.715407985972016,0.698545758784881],[0,0,0,0],[8.999999E+09,8.999999E+09,8.999999E+09,8.999999E+09,8.999999E+09,8.999999E+09]];
	LOCAL CONST Robtarget Tr_meulage_bavure_P16 :=[[81.705078125,97.9371015625,53],[0.00830216452804949,-0.00850110626532978,-0.715377897968694,0.698636721303931],[0,0,0,0],[8.999999E+09,8.999999E+09,8.999999E+09,8.999999E+09,8.999999E+09,8.999999E+09]];
	LOCAL CONST Robtarget Tr_meulage_bavure_P17 :=[[62.0113828125,98.530734375,53],[0.00752660586442575,-0.00770613452821541,-0.715349347414217,0.69868396063517],[0,0,0,0],[8.999999E+09,8.999999E+09,8.999999E+09,8.999999E+09,8.999999E+09,8.999999E+09]];
	LOCAL CONST Robtarget Tr_meulage_bavure_P18 :=[[60.42755078125,98.5550234375,53],[0.00749633052467423,-0.00767462368976842,-0.715326322869143,0.698708205898854],[0,0,0,0],[8.999999E+09,8.999999E+09,8.999999E+09,8.999999E+09,8.999999E+09,8.999999E+09]];
	LOCAL CONST Robtarget Tr_meulage_bavure_P19 :=[[50.404359375,98.8545859375,53],[0.00776030293537024,-0.00794424933743714,-0.715295894944966,0.698733460824438],[0,0,0,0],[8.999999E+09,8.999999E+09,8.999999E+09,8.999999E+09,8.999999E+09,8.999999E+09]];
	LOCAL CONST Robtarget Tr_meulage_bavure_P20 :=[[44.00372265625,99.0664375,53],[0.0080498765807494,-0.00824000643570157,-0.715263703174872,0.698759713135741],[0,0,0,0],[8.999999E+09,8.999999E+09,8.999999E+09,8.999999E+09,8.999999E+09,8.999999E+09]];
	LOCAL CONST Robtarget Tr_meulage_bavure_P21 :=[[32.69549609375,99.2951953125,53],[0.00823528165162698,-0.00842893426962742,-0.715226013097772,0.698793877614466],[0,0,0,0],[8.999999E+09,8.999999E+09,8.999999E+09,8.999999E+09,8.999999E+09,8.999999E+09]];
	LOCAL CONST Robtarget Tr_meulage_bavure_P22 :=[[24.02682421875,99.5107734375,53],[0.00829226989425514,-0.00848606665235417,-0.715176105157706,0.69884359018612],[0,0,0,0],[8.999999E+09,8.999999E+09,8.999999E+09,8.999999E+09,8.999999E+09,8.999999E+09]];
	LOCAL CONST Robtarget Tr_meulage_bavure_P23 :=[[20.713103515625,99.58075,53],[0.00824084790787603,-0.00843176731180318,-0.715107321417406,0.698915239911809],[0,0,0,0],[8.999999E+09,8.999999E+09,8.999999E+09,8.999999E+09,8.999999E+09,8.999999E+09]];
	LOCAL CONST Robtarget Tr_meulage_bavure_P24 :=[[9.33969140625,99.930453125,53],[0.00811897120363269,-0.00830483529774257,-0.715014915558275,0.699012719874585],[0,0,0,0],[8.999999E+09,8.999999E+09,8.999999E+09,8.999999E+09,8.999999E+09,8.999999E+09]];
	LOCAL CONST Robtarget Tr_meulage_bavure_P25 :=[[6.80206298828125,100.0127890625,53],[0.00797402543424442,-0.00815381486444001,-0.714898523302619,0.699135202662021],[0,0,0,0],[8.999999E+09,8.999999E+09,8.999999E+09,8.999999E+09,8.999999E+09,8.999999E+09]];
	LOCAL CONST Robtarget Tr_meulage_bavure_P26 :=[[-6.8071591796875,100.2854609375,53],[0.007846198540718,-0.00801975150823996,-0.714753860537639,0.699286092812339],[0,0,0,0],[8.999999E+09,8.999999E+09,8.999999E+09,8.999999E+09,8.999999E+09,8.999999E+09]];
	LOCAL CONST Robtarget Tr_meulage_bavure_P27 :=[[-7.3994443359375,100.3124375,53],[0.0077710347296564,-0.00793883728488048,-0.714574769262709,0.699470860733269],[0,0,0,0],[8.999999E+09,8.999999E+09,8.999999E+09,8.999999E+09,8.999999E+09,8.999999E+09]];
	LOCAL CONST Robtarget Tr_meulage_bavure_P28 :=[[-15.121642578125,100.5769921875,53],[0.00778383115400197,-0.00794716595952957,-0.714365952841401,0.69968388572753],[0,0,0,0],[8.999999E+09,8.999999E+09,8.999999E+09,8.999999E+09,8.999999E+09,8.999999E+09]];
	LOCAL CONST Robtarget Tr_meulage_bavure_P29 :=[[-19.364501953125,100.651640625,53],[0.00791352162149719,-0.00807398864155508,-0.714122414857029,0.699929541798121],[0,0,0,0],[8.999999E+09,8.999999E+09,8.999999E+09,8.999999E+09,8.999999E+09,8.999999E+09]];
	LOCAL CONST Robtarget Tr_meulage_bavure_P30 :=[[-28.033203125,100.991546875,53],[0.0081646839898892,-0.00832349349697336,-0.713835797572547,0.70021604629951],[0,0,0,0],[8.999999E+09,8.999999E+09,8.999999E+09,8.999999E+09,8.999999E+09,8.999999E+09]];
	LOCAL CONST Robtarget Tr_meulage_bavure_P31 :=[[-31.077423828125,101.018921875,53],[0.0084982210639963,-0.00865553829383419,-0.713509156467974,0.700540894974698],[0,0,0,0],[8.999999E+09,8.999999E+09,8.999999E+09,8.999999E+09,8.999999E+09,8.999999E+09]];
	LOCAL CONST Robtarget Tr_meulage_bavure_P32 :=[[-38.86975,101.2014765625,53],[0.00882966659006116,-0.0089838785724014,-0.713144899741324,0.700903473301882],[0,0,0,0],[8.999999E+09,8.999999E+09,8.999999E+09,8.999999E+09,8.999999E+09,8.999999E+09]];
	LOCAL CONST Robtarget Tr_meulage_bavure_P33 :=[[-42.005921875,101.266296875,53],[0.009053452783813,-0.0092009965929877,-0.712739388133502,0.701310160526331],[0,0,0,0],[8.999999E+09,8.999999E+09,8.999999E+09,8.999999E+09,8.999999E+09,8.999999E+09]];
	LOCAL CONST Robtarget Tr_meulage_bavure_P34 :=[[-42.84326171875,101.2991328125,53],[0.0090821970574109,-0.00921843806055967,-0.712291522492658,0.701764434181032],[0,0,0,0],[8.999999E+09,8.999999E+09,8.999999E+09,8.999999E+09,8.999999E+09,8.999999E+09]];
	LOCAL CONST Robtarget Tr_meulage_bavure_P35 :=[[-44.25528125,101.345546875,53],[0.00888686913738419,-0.00900749002090178,-0.711800028035025,0.702268188635792],[0,0,0,0],[8.999999E+09,8.999999E+09,8.999999E+09,8.999999E+09,8.999999E+09,8.999999E+09]];
	LOCAL CONST Robtarget Tr_meulage_bavure_P36 :=[[-54.80258203125,101.5965859375,53],[0.00850575735048454,-0.00860797712498984,-0.711265531874662,0.702819249870665],[0,0,0,0],[8.999999E+09,8.999999E+09,8.999999E+09,8.999999E+09,8.999999E+09,8.999999E+09]];
	LOCAL CONST Robtarget Tr_meulage_bavure_P37 :=[[-64.728484375,101.8648671875,53],[0.00801723311991166,-0.00810000019877129,-0.710682467859603,0.703420602375894],[0,0,0,0],[8.999999E+09,8.999999E+09,8.999999E+09,8.999999E+09,8.999999E+09,8.999999E+09]];
	LOCAL CONST Robtarget Tr_meulage_bavure_P38 :=[[-71.560609375,102.00265625,53],[0.00750348241737372,-0.00756721990678621,-0.710050627114797,0.70406998364394],[0,0,0,0],[8.999999E+09,8.999999E+09,8.999999E+09,8.999999E+09,8.999999E+09,8.999999E+09]];
	LOCAL CONST Robtarget Tr_meulage_bavure_P39 :=[[-84.2489609375,102.2153046875,53],[0.00700401152365725,-0.00704981324915689,-0.709372460430323,0.70476375924047],[0,0,0,0],[8.999999E+09,8.999999E+09,8.999999E+09,8.999999E+09,8.999999E+09,8.999999E+09]];
	LOCAL CONST Robtarget Tr_meulage_bavure_P40 :=[[-84.6449296875,102.2199375,53],[0.00643723901908446,-0.00646589282097475,-0.708645798052384,0.705505412513992],[0,0,0,0],[8.999999E+09,8.999999E+09,8.999999E+09,8.999999E+09,8.999999E+09,8.999999E+09]];
	LOCAL CONST Robtarget Tr_meulage_bavure_P41 :=[[-84.70978125,102.2224765625,53],[0.00560290700908717,-0.00561548790906787,-0.707877049810515,0.706291127000866],[0,0,0,0],[8.999999E+09,8.999999E+09,8.999999E+09,8.999999E+09,8.999999E+09,8.999999E+09]];
	LOCAL CONST Robtarget Tr_meulage_bavure_P42 :=[[-84.8934609375,102.2269296875,53],[0.00411893326035562,-0.00411866501651484,-0.707071759613592,0.70711781037124],[0,0,0,0],[8.999999E+09,8.999999E+09,8.999999E+09,8.999999E+09,8.999999E+09,8.999999E+09]];
	LOCAL CONST Robtarget Tr_meulage_bavure_P43 :=[[-90.20971875,102.410671875,53],[0.00134230635421909,-0.00133901670844186,-0.706237449302047,0.707972506847014],[0,0,0,0],[8.999999E+09,8.999999E+09,8.999999E+09,8.999999E+09,8.999999E+09,8.999999E+09]];
	LOCAL CONST Robtarget Tr_meulage_bavure_P44 :=[[-94.9345078125,102.46353125,53],[0.00359143227307249,-0.00357395375205285,0.70537078340552,-0.708820418996722],[0,0,0,0],[8.999999E+09,8.999999E+09,8.999999E+09,8.999999E+09,8.999999E+09,8.999999E+09]];
	LOCAL CONST Robtarget Tr_meulage_bavure_P45 :=[[-99.332609375,102.491609375,53],[0.0118382103799242,-0.0117518089065671,0.704414164943357,-0.709593148212113],[0,0,0,0],[8.999999E+09,8.999999E+09,8.999999E+09,8.999999E+09,8.999999E+09,8.999999E+09]];
	LOCAL CONST Robtarget Tr_meulage_bavure_P46 :=[[-102.443421875,102.53921875,53],[0.0247368002260729,-0.0244972451477689,0.703231371194898,-0.710108170817721],[0,0,0,0],[8.999999E+09,8.999999E+09,8.999999E+09,8.999999E+09,8.999999E+09,8.999999E+09]];
	LOCAL CONST Robtarget Tr_meulage_bavure_P47 :=[[-104.810546875,102.651125,53],[0.0437252578300974,-0.0432020619374765,0.701509106045304,-0.710004688581393],[0,0,0,0],[8.999999E+09,8.999999E+09,8.999999E+09,8.999999E+09,8.999999E+09,8.999999E+09]];
	LOCAL CONST Robtarget Tr_meulage_bavure_P48 :=[[-107.8382265625,102.594421875,53],[0.0701514161662176,-0.0691619482538018,0.698651931167532,-0.708647220272183],[0,0,0,0],[8.999999E+09,8.999999E+09,8.999999E+09,8.999999E+09,8.999999E+09,8.999999E+09]];
	LOCAL CONST Robtarget Tr_meulage_bavure_P49 :=[[-108.137484375,102.604953125,53],[0.104851901093992,-0.103172073529582,0.693744107348957,-0.705039513502031],[0,0,0,0],[8.999999E+09,8.999999E+09,8.999999E+09,8.999999E+09,8.999999E+09,8.999999E+09]];
	LOCAL CONST Robtarget Tr_meulage_bavure_P50 :=[[-108.5615859375,102.5401015625,53],[0.147610392114513,-0.145002810486695,0.685611794264447,-0.697941132658224],[0,0,0,0],[8.999999E+09,8.999999E+09,8.999999E+09,8.999999E+09,8.999999E+09,8.999999E+09]];
	LOCAL CONST Robtarget Tr_meulage_bavure_P51 :=[[-112.5101953125,101.8948359375,53],[0.19640588313291,-0.192677049948771,0.673270219403821,-0.686299858048762],[0,0,0,0],[8.999999E+09,8.999999E+09,8.999999E+09,8.999999E+09,8.999999E+09,8.999999E+09]];
	LOCAL CONST Robtarget Tr_meulage_bavure_P52 :=[[-114.612578125,100.509796875,53],[0.247372828449912,-0.242440541310549,0.656623086276101,-0.669981634257975],[0,0,0,0],[8.999999E+09,8.999999E+09,8.999999E+09,8.999999E+09,8.999999E+09,8.999999E+09]];
	LOCAL CONST Robtarget Tr_meulage_bavure_P53 :=[[-115.32415625,100.02740625,53],[0.296021364616972,-0.289959945554678,0.636851857352569,-0.650164820219317],[0,0,0,0],[8.999999E+09,8.999999E+09,8.999999E+09,8.999999E+09,8.999999E+09,8.999999E+09]];
	LOCAL CONST Robtarget Tr_meulage_bavure_P54 :=[[-115.9504375,99.0186171875,53],[0.339059081634174,-0.332086971390644,0.615898530028053,-0.628829216324483],[0,0,0,0],[8.999999E+09,8.999999E+09,8.999999E+09,8.999999E+09,8.999999E+09,8.999999E+09]];
	LOCAL CONST Robtarget Tr_meulage_bavure_P55 :=[[-116.7562578125,97.1141640625,53],[0.375324714878579,-0.367747459832277,0.59545416845373,-0.607723207932113],[0,0,0,0],[8.999999E+09,8.999999E+09,8.999999E+09,8.999999E+09,8.999999E+09,8.999999E+09]];
	LOCAL CONST Robtarget Tr_meulage_bavure_P56 :=[[-117.1447421875,95.895875,53],[0.405266452411773,-0.397424249497356,0.576441674901934,-0.587816352186031],[0,0,0,0],[8.999999E+09,8.999999E+09,8.999999E+09,8.999999E+09,8.999999E+09,8.999999E+09]];
	LOCAL CONST Robtarget Tr_meulage_bavure_P57 :=[[-117.186734375,95.1318984375,53],[0.429845330397908,-0.422084458555267,0.559227780568614,-0.569510308266253],[0,0,0,0],[8.999999E+09,8.999999E+09,8.999999E+09,8.999999E+09,8.999999E+09,8.999999E+09]];
	LOCAL CONST Robtarget Tr_meulage_bavure_P58 :=[[-117.481078125,89.1402578125,53],[0.449817909399474,-0.442474913414983,0.544047012214227,-0.553075625825857],[0,0,0,0],[8.999999E+09,8.999999E+09,8.999999E+09,8.999999E+09,8.999999E+09,8.999999E+09]];
	LOCAL CONST Robtarget Tr_meulage_bavure_P59 :=[[-117.48034375,84.272859375,53],[0.465525143591152,-0.45891557199203,0.531269289015285,-0.538920941341919],[0,0,0,0],[8.999999E+09,8.999999E+09,8.999999E+09,8.999999E+09,8.999999E+09,8.999999E+09]];
	LOCAL CONST Robtarget Tr_meulage_bavure_P60 :=[[-117.52490625,81.8545546875,53],[0.477153267311431,-0.471551785543213,0.52128185711092,-0.527474073762895],[0,0,0,0],[8.999999E+09,8.999999E+09,8.999999E+09,8.999999E+09,8.999999E+09,8.999999E+09]];
	LOCAL CONST Robtarget Tr_meulage_bavure_P61 :=[[-117.6038828125,77.18375,53],[0.484989427629277,-0.480631089490895,0.514276518492805,-0.518939951660634],[0,0,0,0],[8.999999E+09,8.999999E+09,8.999999E+09,8.999999E+09,8.999999E+09,8.999999E+09]];
	LOCAL CONST Robtarget Tr_meulage_bavure_P62 :=[[-117.78140625,71.7738671875,53],[0.489546841809786,-0.48660043509609,0.510099637520675,-0.513188333888872],[0,0,0,0],[8.999999E+09,8.999999E+09,8.999999E+09,8.999999E+09,8.999999E+09,8.999999E+09]];
	LOCAL CONST Robtarget Tr_meulage_bavure_P63 :=[[-117.858828125,65.2600078125,53],[0.491562696682377,-0.490129310724038,0.508245161411448,-0.509731527278213],[0,0,0,0],[8.999999E+09,8.999999E+09,8.999999E+09,8.999999E+09,8.999999E+09,8.999999E+09]];
	LOCAL CONST Robtarget Tr_meulage_bavure_P64 :=[[-117.9099765625,63.17498828125,53],[0.491797868420598,-0.491931700505519,0.508074057240477,-0.507935833559619],[0,0,0,0],[8.999999E+09,8.999999E+09,8.999999E+09,8.999999E+09,8.999999E+09,8.999999E+09]];
	LOCAL CONST Robtarget Tr_meulage_bavure_P65 :=[[-117.9591640625,61.1898515625,53],[0.490966917520564,-0.492665661716015,0.508927845106439,-0.507173027813579],[0,0,0,0],[8.999999E+09,8.999999E+09,8.999999E+09,8.999999E+09,8.999999E+09,8.999999E+09]];
	LOCAL CONST Robtarget Tr_meulage_bavure_P66 :=[[-118.0036015625,59.44287109375,53],[0.489629997552147,-0.49285865314003,0.510271020092207,-0.506928298259367],[0,0,0,0],[8.999999E+09,8.999999E+09,8.999999E+09,8.999999E+09,8.999999E+09,8.999999E+09]];
	LOCAL CONST Robtarget Tr_meulage_bavure_P67 :=[[-118.0876484375,57.84430078125,53],[0.488176148008532,-0.492869115024469,0.511726065038389,-0.506853547221359],[0,0,0,0],[8.999999E+09,8.999999E+09,8.999999E+09,8.999999E+09,8.999999E+09,8.999999E+09]];
	LOCAL CONST Robtarget Tr_meulage_bavure_P68 :=[[-118.232359375,52.42559765625,53],[0.486850551472581,-0.492912688805498,0.51305379209608,-0.506743947335546],[0,0,0,0],[8.999999E+09,8.999999E+09,8.999999E+09,8.999999E+09,8.999999E+09,8.999999E+09]];
	LOCAL CONST Robtarget Tr_meulage_bavure_P69 :=[[-118.43503125,48.23135546875,53],[0.485742161712944,-0.493075058097905,0.514167439379026,-0.506520862056637],[0,0,0,0],[8.999999E+09,8.999999E+09,8.999999E+09,8.999999E+09,8.999999E+09,8.999999E+09]];
	LOCAL CONST Robtarget Tr_meulage_bavure_P70 :=[[-118.5796171875,42.5523671875,53],[0.484876266208668,-0.493362386913663,0.515041552286503,-0.506182537297272],[0,0,0,0],[8.999999E+09,8.999999E+09,8.999999E+09,8.999999E+09,8.999999E+09,8.999999E+09]];
	LOCAL CONST Robtarget Tr_meulage_bavure_P71 :=[[-118.759734375,35.33465625,53],[0.484244798308208,-0.493759326858851,0.515683354634348,-0.505746359556253],[0,0,0,0],[8.999999E+09,8.999999E+09,8.999999E+09,8.999999E+09,8.999999E+09,8.999999E+09]];
	LOCAL CONST Robtarget Tr_meulage_bavure_P72 :=[[-118.944515625,29.635986328125,53],[0.483846576346188,-0.4942738926872,0.516093666004055,-0.505206034679326],[0,0,0,0],[8.999999E+09,8.999999E+09,8.999999E+09,8.999999E+09,8.999999E+09,8.999999E+09]];
	LOCAL CONST Robtarget Tr_meulage_bavure_P73 :=[[-119.1793203125,25.164306640625,53],[0.483707809771266,-0.494929134704558,0.516245991738784,-0.504541358463824],[0,0,0,0],[8.999999E+09,8.999999E+09,8.999999E+09,8.999999E+09,8.999999E+09,8.999999E+09]];
	LOCAL CONST Robtarget Tr_meulage_bavure_P74 :=[[-119.5641484375,19.09484765625,53],[0.483856473877286,-0.495763644787542,0.516111905539518,-0.503716013398798],[0,0,0,0],[8.999999E+09,8.999999E+09,8.999999E+09,8.999999E+09,8.999999E+09,8.999999E+09]];
	LOCAL CONST Robtarget Tr_meulage_bavure_P75 :=[[-119.903109375,6.8254091796875,53],[0.484306432188968,-0.496794593552821,0.515676052358436,-0.502713258807741],[0,0,0,0],[8.999999E+09,8.999999E+09,8.999999E+09,8.999999E+09,8.999999E+09,8.999999E+09]];
	LOCAL CONST Robtarget Tr_meulage_bavure_P76 :=[[-120.0164453125,3.00881958007813,53],[0.485016421593797,-0.498005604936774,0.514977313075621,-0.501545466785734],[0,0,0,0],[8.999999E+09,8.999999E+09,8.999999E+09,8.999999E+09,8.999999E+09,8.999999E+09]];
	LOCAL CONST Robtarget Tr_meulage_bavure_P77 :=[[-120.199796875,-6.6208798828125,53],[0.485902476213176,-0.49932460341703,0.51409706944718,-0.500277850017518],[0,0,0,0],[8.999999E+09,8.999999E+09,8.999999E+09,8.999999E+09,8.999999E+09,8.999999E+09]];
	LOCAL CONST Robtarget Tr_meulage_bavure_P78 :=[[-120.2404765625,-7.885498046875,53],[0.486833037627381,-0.50061696132582,0.513165713085078,-0.49903627365281],[0,0,0,0],[8.999999E+09,8.999999E+09,8.999999E+09,8.999999E+09,8.999999E+09,8.999999E+09]];
	LOCAL CONST Robtarget Tr_meulage_bavure_P79 :=[[-120.73815625,-17.822693359375,53],[0.487631181735516,-0.501725052410663,0.512361764650172,-0.497969099952299],[0,0,0,0],[8.999999E+09,8.999999E+09,8.999999E+09,8.999999E+09,8.999999E+09,8.999999E+09]];
	LOCAL CONST Robtarget Tr_meulage_bavure_P80 :=[[-120.7496953125,-19.84973046875,53],[0.488143444420689,-0.502502522575657,0.511842585063545,-0.497216613348424],[0,0,0,0],[8.999999E+09,8.999999E+09,8.999999E+09,8.999999E+09,8.999999E+09,8.999999E+09]];
	LOCAL CONST Robtarget Tr_meulage_bavure_P81 :=[[-120.699125,-21.677947265625,53],[0.488285823796737,-0.502872127315487,0.511696066000183,-0.496853815410807],[0,0,0,0],[8.999999E+09,8.999999E+09,8.999999E+09,8.999999E+09,8.999999E+09,8.999999E+09]];
	LOCAL CONST Robtarget Tr_meulage_bavure_P82 :=[[-120.797671875,-28.73162890625,53],[0.488085153715985,-0.502876919728709,0.511896621183714,-0.496839547084274],[0,0,0,0],[8.999999E+09,8.999999E+09,8.999999E+09,8.999999E+09,8.999999E+09,8.999999E+09]];
	LOCAL CONST Robtarget Tr_meulage_bavure_P83 :=[[-120.925171875,-34.84551953125,53],[0.487685624066883,-0.502659166518369,0.512298576427172,-0.497037888881971],[0,0,0,0],[8.999999E+09,8.999999E+09,8.999999E+09,8.999999E+09,8.999999E+09,8.999999E+09]];
	LOCAL CONST Robtarget Tr_meulage_bavure_P84 :=[[-120.9287109375,-35.01052734375,53],[0.487250745864966,-0.502401275267404,0.512736109163196,-0.497273920112354],[0,0,0,0],[8.999999E+09,8.999999E+09,8.999999E+09,8.999999E+09,8.999999E+09,8.999999E+09]];
	LOCAL CONST Robtarget Tr_meulage_bavure_P85 :=[[-121.3921796875,-50.7028359375,53],[0.486910553511978,-0.502234847352085,0.513077868183531,-0.497422729842666],[0,0,0,0],[8.999999E+09,8.999999E+09,8.999999E+09,8.999999E+09,8.999999E+09,8.999999E+09]];
	LOCAL CONST Robtarget Tr_meulage_bavure_P86 :=[[-121.42321875,-53.91790625,53],[0.486694754960823,-0.502189555282366,0.513294044643069,-0.497456621016229],[0,0,0,0],[8.999999E+09,8.999999E+09,8.999999E+09,8.999999E+09,8.999999E+09,8.999999E+09]];
	LOCAL CONST Robtarget Tr_meulage_bavure_P87 :=[[-121.621765625,-67.8473515625,53],[0.486539025412648,-0.502201889671758,0.513449617455106,-0.497435954767879],[0,0,0,0],[8.999999E+09,8.999999E+09,8.999999E+09,8.999999E+09,8.999999E+09,8.999999E+09]];
	LOCAL CONST Robtarget Tr_meulage_bavure_P88 :=[[-121.64196875,-68.861203125,53],[0.486347004848985,-0.50215671669117,0.513642015738386,-0.49747070509184],[0,0,0,0],[8.999999E+09,8.999999E+09,8.999999E+09,8.999999E+09,8.999999E+09,8.999999E+09]];
	LOCAL CONST Robtarget Tr_meulage_bavure_P89 :=[[-121.7797265625,-73.7997890625,53],[0.486043194759845,-0.501974341257085,0.513947395724476,-0.497636260711764],[0,0,0,0],[8.999999E+09,8.999999E+09,8.999999E+09,8.999999E+09,8.999999E+09,8.999999E+09]];
	LOCAL CONST Robtarget Tr_meulage_bavure_P90 :=[[-121.9932578125,-79.1463203125,53],[0.485619550864874,-0.501638970147616,0.514373635804569,-0.497947545667439],[0,0,0,0],[8.999999E+09,8.999999E+09,8.999999E+09,8.999999E+09,8.999999E+09,8.999999E+09]];
	LOCAL CONST Robtarget Tr_meulage_bavure_P91 :=[[-122.0453515625,-85.0171015625,53],[0.485153816425883,-0.50122172241152,0.514842024154476,-0.498337485600624],[0,0,0,0],[8.999999E+09,8.999999E+09,8.999999E+09,8.999999E+09,8.999999E+09,8.999999E+09]];
	LOCAL CONST Robtarget Tr_meulage_bavure_P92 :=[[-122.0739453125,-85.9891171875,53],[0.484869259510317,-0.500951057478073,0.51512795565244,-0.498591043339986],[0,0,0,0],[8.999999E+09,8.999999E+09,8.999999E+09,8.999999E+09,8.999999E+09,8.999999E+09]];
	LOCAL CONST Robtarget Tr_meulage_bavure_P93 :=[[-122.286984375,-91.65625,53],[0.485142785405193,-0.501210083451084,0.514853120162396,-0.498348467114421],[0,0,0,0],[8.999999E+09,8.999999E+09,8.999999E+09,8.999999E+09,8.999999E+09,8.999999E+09]];
	LOCAL CONST Robtarget Tr_meulage_bavure_P94 :=[[-122.3317265625,-93.0854921875,53],[0.486579448856203,-0.502615245138622,0.513404924969787,-0.497024887024588],[0,0,0,0],[8.999999E+09,8.999999E+09,8.999999E+09,8.999999E+09,8.999999E+09,8.999999E+09]];
	LOCAL CONST Robtarget Tr_meulage_bavure_P95 :=[[-122.358125,-94.2397734375,53],[0.489973723479603,-0.505989546897738,0.509952113625751,-0.49381086514817],[0,0,0,0],[8.999999E+09,8.999999E+09,8.999999E+09,8.999999E+09,8.999999E+09,8.999999E+09]];
	LOCAL CONST Robtarget Tr_meulage_bavure_P96 :=[[-122.58590625,-97.7452109375,53],[0.496208595119145,-0.512242162399172,0.503490969071187,-0.487731320764068],[0,0,0,0],[8.999999E+09,8.999999E+09,8.999999E+09,8.999999E+09,8.999999E+09,8.999999E+09]];
	LOCAL CONST Robtarget Tr_meulage_bavure_P97 :=[[-122.634796875,-102.9755234375,53],[0.506105461811494,-0.522219356804991,0.492902769705262,-0.477693483857208],[0,0,0,0],[8.999999E+09,8.999999E+09,8.999999E+09,8.999999E+09,8.999999E+09,8.999999E+09]];
	LOCAL CONST Robtarget Tr_meulage_bavure_P98 :=[[-122.68484375,-105.89503125,53],[0.520139901059478,-0.53640428565838,0.477138073990327,-0.462670707957573],[0,0,0,0],[8.999999E+09,8.999999E+09,8.999999E+09,8.999999E+09,8.999999E+09,8.999999E+09]];
	LOCAL CONST Robtarget Tr_meulage_bavure_P99 :=[[-122.785640625,-110.49609375,53],[0.538324535147367,-0.554808810283245,0.455262116686808,-0.441735536266111],[0,0,0,0],[8.999999E+09,8.999999E+09,8.999999E+09,8.999999E+09,8.999999E+09,8.999999E+09]];
	LOCAL CONST Robtarget Tr_meulage_bavure_P100 :=[[-122.9415,-114.1469609375,53],[0.560200657550605,-0.576950741547481,0.426444028351166,-0.414063468312904],[0,0,0,0],[8.999999E+09,8.999999E+09,8.999999E+09,8.999999E+09,8.999999E+09,8.999999E+09]];
	LOCAL CONST Robtarget Tr_meulage_bavure_P101 :=[[-122.8875703125,-115.18109375,53],[0.58489483386865,-0.601921759587707,0.389915328353179,-0.378885557080018],[0,0,0,0],[8.999999E+09,8.999999E+09,8.999999E+09,8.999999E+09,8.999999E+09,8.999999E+09]];
	LOCAL CONST Robtarget Tr_meulage_bavure_P102 :=[[-121.8850390625,-117.89328125,53],[0.61107106859449,-0.628350975419892,0.345129322422154,-0.335638125992987],[0,0,0,0],[8.999999E+09,8.999999E+09,8.999999E+09,8.999999E+09,8.999999E+09,8.999999E+09]];
	LOCAL CONST Robtarget Tr_meulage_bavure_P103 :=[[-121.3135390625,-119.283921875,53],[0.636707084007005,-0.654145166350946,0.292575810643022,-0.284776378131277],[0,0,0,0],[8.999999E+09,8.999999E+09,8.999999E+09,8.999999E+09,8.999999E+09,8.999999E+09]];
	LOCAL CONST Robtarget Tr_meulage_bavure_P104 :=[[-120.65228125,-120.3115390625,53],[0.659118620795482,-0.676557604606763,0.235210284855991,-0.229147492387293],[0,0,0,0],[8.999999E+09,8.999999E+09,8.999999E+09,8.999999E+09,8.999999E+09,8.999999E+09]];
	LOCAL CONST Robtarget Tr_meulage_bavure_P105 :=[[-118.755375,-121.54021875,53],[0.675955878075704,-0.693184266960163,0.179100373936449,-0.174649016572179],[0,0,0,0],[8.999999E+09,8.999999E+09,8.999999E+09,8.999999E+09,8.999999E+09,8.999999E+09]];
	LOCAL CONST Robtarget Tr_meulage_bavure_P106 :=[[-118.17196875,-121.7504140625,53],[0.686609551685376,-0.703408383814174,0.131530283625081,-0.128389071200956],[0,0,0,0],[8.999999E+09,8.999999E+09,8.999999E+09,8.999999E+09,8.999999E+09,8.999999E+09]];
	LOCAL CONST Robtarget Tr_meulage_bavure_P107 :=[[-117.1280859375,-121.8553046875,53],[0.692293599145889,-0.708492469044411,0.0979847101073754,-0.0957444017901753],[0,0,0,0],[8.999999E+09,8.999999E+09,8.999999E+09,8.999999E+09,8.999999E+09,8.999999E+09]];
	LOCAL CONST Robtarget Tr_meulage_bavure_P108 :=[[-114.791625,-122.3441953125,53],[0.694791302491848,-0.710265308539386,0.0808389731699252,-0.0790777964030625],[0,0,0,0],[8.999999E+09,8.999999E+09,8.999999E+09,8.999999E+09,8.999999E+09,8.999999E+09]];
	LOCAL CONST Robtarget Tr_meulage_bavure_P109 :=[[-109.6820390625,-121.9300078125,53],[0.695255241777794,-0.709918659077907,0.0803098100735338,-0.0786510055846779],[0,0,0,0],[8.999999E+09,8.999999E+09,8.999999E+09,8.999999E+09,8.999999E+09,8.999999E+09]];
	LOCAL CONST Robtarget Tr_meulage_bavure_P110 :=[[-107.252625,-121.83384375,53],[0.693816496758844,-0.707583792110326,0.0956461475101601,-0.0937851823825156],[0,0,0,0],[8.999999E+09,8.999999E+09,8.999999E+09,8.999999E+09,8.999999E+09,8.999999E+09]];
	LOCAL CONST Robtarget Tr_meulage_bavure_P111 :=[[-104.9573046875,-122.360609375,53],[0.689634615978067,-0.702402069829033,0.125707360744124,-0.123422397478828],[0,0,0,0],[8.999999E+09,8.999999E+09,8.999999E+09,8.999999E+09,8.999999E+09,8.999999E+09]];
	LOCAL CONST Robtarget Tr_meulage_bavure_P112 :=[[-103.8669140625,-122.6539140625,53],[0.681188491058003,-0.69284841816526,0.168660455278171,-0.165822073082498],[0,0,0,0],[8.999999E+09,8.999999E+09,8.999999E+09,8.999999E+09,8.999999E+09,8.999999E+09]];
	LOCAL CONST Robtarget Tr_meulage_bavure_P113 :=[[-102.1970546875,-123.70884375,53],[0.666984449278629,-0.677421308855816,0.221049947439571,-0.217644286544628],[0,0,0,0],[8.999999E+09,8.999999E+09,8.999999E+09,8.999999E+09,8.999999E+09,8.999999E+09]];
	LOCAL CONST Robtarget Tr_meulage_bavure_P114 :=[[-101.2503984375,-124.348828125,53],[0.64674989636993,-0.655876537506103,0.277185789090659,-0.273328698494467],[0,0,0,0],[8.999999E+09,8.999999E+09,8.999999E+09,8.999999E+09,8.999999E+09,8.999999E+09]];
	LOCAL CONST Robtarget Tr_meulage_bavure_P115 :=[[-99.53771875,-126.6721328125,53],[0.622386829587385,-0.630177767920647,0.330296426621183,-0.326212945383827],[0,0,0,0],[8.999999E+09,8.999999E+09,8.999999E+09,8.999999E+09,8.999999E+09,8.999999E+09]];
	LOCAL CONST Robtarget Tr_meulage_bavure_P116 :=[[-99.156890625,-127.369953125,53],[0.597220929071256,-0.603717861658887,0.375412391101257,-0.371372376464545],[0,0,0,0],[8.999999E+09,8.999999E+09,8.999999E+09,8.999999E+09,8.999999E+09,8.999999E+09]];
	LOCAL CONST Robtarget Tr_meulage_bavure_P117 :=[[-98.74475,-128.4476953125,53],[0.574157216005002,-0.579451358343486,0.410883472877657,-0.407129446661956],[0,0,0,0],[8.999999E+09,8.999999E+09,8.999999E+09,8.999999E+09,8.999999E+09,8.999999E+09]];
	LOCAL CONST Robtarget Tr_meulage_bavure_P118 :=[[-98.7053828125,-128.6214765625,53],[0.554552468211008,-0.558739640053146,0.437688283473972,-0.434408265510647],[0,0,0,0],[8.999999E+09,8.999999E+09,8.999999E+09,8.999999E+09,8.999999E+09,8.999999E+09]];
	LOCAL CONST Robtarget Tr_meulage_bavure_P119 :=[[-98.5738515625,-130.3565546875,53],[0.538452693013544,-0.541627564170789,0.457798026873148,-0.455114541305738],[0,0,0,0],[8.999999E+09,8.999999E+09,8.999999E+09,8.999999E+09,8.999999E+09,8.999999E+09]];
	LOCAL CONST Robtarget Tr_meulage_bavure_P120 :=[[-98.1612265625,-133.2596875,53],[0.52532644546798,-0.527575727651452,0.473075163963813,-0.471058241118473],[0,0,0,0],[8.999999E+09,8.999999E+09,8.999999E+09,8.999999E+09,8.999999E+09,8.999999E+09]];
	LOCAL CONST Robtarget Tr_meulage_bavure_P121 :=[[-98.3329140625,-138.09928125,53],[0.514677737575522,-0.516082593877863,0.484790352446246,-0.483470678444395],[0,0,0,0],[8.999999E+09,8.999999E+09,8.999999E+09,8.999999E+09,8.999999E+09,8.999999E+09]];
	LOCAL CONST Robtarget Tr_meulage_bavure_P122 :=[[-98.4911484375,-145.174671875,53],[0.506270642638317,-0.506909887853185,0.493632752740732,-0.493010250827368],[0,0,0,0],[8.999999E+09,8.999999E+09,8.999999E+09,8.999999E+09,8.999999E+09,8.999999E+09]];
	LOCAL CONST Robtarget Tr_meulage_bavure_P123 :=[[-98.63678125,-147.956328125,53],[0.500082273558878,-0.500026216072649,0.499917725065847,-0.499973770389248],[0,0,0,0],[8.999999E+09,8.999999E+09,8.999999E+09,8.999999E+09,8.999999E+09,8.999999E+09]];
	LOCAL CONST Robtarget Tr_meulage_bavure_P124 :=[[-98.703640625,-150.04303125,53],[0.49620399122672,-0.49552228324167,0.503756163069623,-0.504449198701917],[0,0,0,0],[8.999999E+09,8.999999E+09,8.999999E+09,8.999999E+09,8.999999E+09,8.999999E+09]];
	LOCAL CONST Robtarget Tr_meulage_bavure_P125 :=[[-98.7443203125,-151.6001875,53],[0.494866641703798,-0.49362898326693,0.505052835064494,-0.50631913611968],[0,0,0,0],[8.999999E+09,8.999999E+09,8.999999E+09,8.999999E+09,8.999999E+09,8.999999E+09]];
	LOCAL CONST Robtarget Tr_meulage_bavure_P126 :=[[-99.13425,-162.702625,53],[0.4965068112055,-0.494770830936712,0.503438749879756,-0.505205142887767],[0,0,0,0],[8.999999E+09,8.999999E+09,8.999999E+09,8.999999E+09,8.999999E+09,8.999999E+09]];
	LOCAL CONST Robtarget Tr_meulage_bavure_P127 :=[[-99.2074921875,-163.42734375,53],[0.501835982690199,-0.499650423229874,0.498163777593295,-0.500342834202258],[0,0,0,0],[8.999999E+09,8.999999E+09,8.999999E+09,8.999999E+09,8.999999E+09,8.999999E+09]];
	LOCAL CONST Robtarget Tr_meulage_bavure_P128 :=[[-99.23184375,-163.845203125,53],[0.511816015565931,-0.509221026600133,0.488008647097737,-0.490495537835317],[0,0,0,0],[8.999999E+09,8.999999E+09,8.999999E+09,8.999999E+09,8.999999E+09,8.999999E+09]];
	LOCAL CONST Robtarget Tr_meulage_bavure_P129 :=[[-99.43228125,-166.61490625,53],[0.527424862127458,-0.52444692148167,0.471300713060767,-0.473976876257316],[0,0,0,0],[8.999999E+09,8.999999E+09,8.999999E+09,8.999999E+09,8.999999E+09,8.999999E+09]];
	LOCAL CONST Robtarget Tr_meulage_bavure_P130 :=[[-99.4632265625,-169.16525,53],[0.549241910004736,-0.54589502711709,0.446029725522727,-0.448764334159147],[0,0,0,0],[8.999999E+09,8.999999E+09,8.999999E+09,8.999999E+09,8.999999E+09,8.999999E+09]];
	LOCAL CONST Robtarget Tr_meulage_bavure_P131 :=[[-99.1395234375,-171.96653125,53],[0.57676816559263,-0.573067190653651,0.410335629025877,-0.412985653149335],[0,0,0,0],[8.999999E+09,8.999999E+09,8.999999E+09,8.999999E+09,8.999999E+09,8.999999E+09]];
	LOCAL CONST Robtarget Tr_meulage_bavure_P132 :=[[-98.85284375,-173.37728125,53],[0.607807159152078,-0.603782738978928,0.363489804731493,-0.36591258963152],[0,0,0,0],[8.999999E+09,8.999999E+09,8.999999E+09,8.999999E+09,8.999999E+09,8.999999E+09]];
	LOCAL CONST Robtarget Tr_meulage_bavure_P133 :=[[-96.9436015625,-175.908484375,53],[0.638435170810813,-0.634138282225533,0.307395742786899,-0.309478640626956],[0,0,0,0],[8.999999E+09,8.999999E+09,8.999999E+09,8.999999E+09,8.999999E+09,8.999999E+09]];
	LOCAL CONST Robtarget Tr_meulage_bavure_P134 :=[[-96.269015625,-176.766796875,53],[0.6644181601609,-0.659929160319348,0.247192128153014,-0.248873589574684],[0,0,0,0],[8.999999E+09,8.999999E+09,8.999999E+09,8.999999E+09,8.999999E+09,8.999999E+09]];
	LOCAL CONST Robtarget Tr_meulage_bavure_P135 :=[[-95.9788515625,-176.893828125,53],[0.683375247840877,-0.678791806437653,0.189411999829264,-0.190690976378556],[0,0,0,0],[8.999999E+09,8.999999E+09,8.999999E+09,8.999999E+09,8.999999E+09,8.999999E+09]];
	LOCAL CONST Robtarget Tr_meulage_bavure_P136 :=[[-93.3845234375,-177.750046875,53],[0.695476369298222,-0.69088558859908,0.139160888785355,-0.140085581864576],[0,0,0,0],[8.999999E+09,8.999999E+09,8.999999E+09,8.999999E+09,8.999999E+09,8.999999E+09]];
	LOCAL CONST Robtarget Tr_meulage_bavure_P137 :=[[-92.5167578125,-177.8825625,53],[0.702382010601795,-0.697853597302292,0.0988248647298706,-0.0994661451266391],[0,0,0,0],[8.999999E+09,8.999999E+09,8.999999E+09,8.999999E+09,8.999999E+09,8.999999E+09]];
	LOCAL CONST Robtarget Tr_meulage_bavure_P138 :=[[-89.7932421875,-178.170375,53],[0.705967208174932,-0.70154499047964,0.0685039359035387,-0.0689357532804153],[0,0,0,0],[8.999999E+09,8.999999E+09,8.999999E+09,8.999999E+09,8.999999E+09,8.999999E+09]];
	LOCAL CONST Robtarget Tr_meulage_bavure_P139 :=[[-88.46340625,-178.1251875,53],[0.707672285378205,-0.703382458267663,0.0470424180845782,-0.0473293229370844],[0,0,0,0],[8.999999E+09,8.999999E+09,8.999999E+09,8.999999E+09,8.999999E+09,8.999999E+09]];
	LOCAL CONST Robtarget Tr_meulage_bavure_P140 :=[[-86.160890625,-178.04278125,53],[0.708410000644529,-0.704271928057089,0.0327390417603778,-0.032931405712213],[0,0,0,0],[8.999999E+09,8.999999E+09,8.999999E+09,8.999999E+09,8.999999E+09,8.999999E+09]];
	LOCAL CONST Robtarget Tr_meulage_bavure_P141 :=[[-83.5302109375,-178.12178125,53],[0.708690694549774,-0.704714242369941,0.0237586598455544,-0.0238927215248176],[0,0,0,0],[8.999999E+09,8.999999E+09,8.999999E+09,8.999999E+09,8.999999E+09,8.999999E+09]];
	LOCAL CONST Robtarget Tr_meulage_bavure_P142 :=[[-80.8863203125,-178.19215625,53],[0.708769423852601,-0.704956922861315,0.0184114677012428,-0.0185110393723417],[0,0,0,0],[8.999999E+09,8.999999E+09,8.999999E+09,8.999999E+09,8.999999E+09,8.999999E+09]];
	LOCAL CONST Robtarget Tr_meulage_bavure_P143 :=[[-76.229828125,-178.44328125,53],[0.70876368862497,-0.705112524815751,0.0152959430937564,-0.0153751474645288],[0,0,0,0],[8.999999E+09,8.999999E+09,8.999999E+09,8.999999E+09,8.999999E+09,8.999999E+09]];
	LOCAL CONST Robtarget Tr_meulage_bavure_P144 :=[[-70.754640625,-178.6341875,53],[0.708719910332434,-0.705231657513315,0.013464768717618,-0.0135313688438852],[0,0,0,0],[8.999999E+09,8.999999E+09,8.999999E+09,8.999999E+09,8.999999E+09,8.999999E+09]];
	LOCAL CONST Robtarget Tr_meulage_bavure_P145 :=[[-63.199828125,-178.86859375,53],[0.708658494082314,-0.705334555900041,0.0123463141298838,-0.0124044969944597],[0,0,0,0],[8.999999E+09,8.999999E+09,8.999999E+09,8.999999E+09,8.999999E+09,8.999999E+09]];
	LOCAL CONST Robtarget Tr_meulage_bavure_P146 :=[[-57.44149609375,-178.94209375,53],[0.708591084679327,-0.70542735519092,0.0116126858898536,-0.0116647669390488],[0,0,0,0],[8.999999E+09,8.999999E+09,8.999999E+09,8.999999E+09,8.999999E+09,8.999999E+09]];
	LOCAL CONST Robtarget Tr_meulage_bavure_P147 :=[[-53.23828125,-179.08309375,53],[0.708518385474508,-0.705515393439044,0.0111504792765129,-0.0111979407504515],[0,0,0,0],[8.999999E+09,8.999999E+09,8.999999E+09,8.999999E+09,8.999999E+09,8.999999E+09]];
	LOCAL CONST Robtarget Tr_meulage_bavure_P148 :=[[-43.2679765625,-179.266203125,53],[0.708439374459743,-0.705602387927693,0.0109078909427208,-0.0109517478516925],[0,0,0,0],[8.999999E+09,8.999999E+09,8.999999E+09,8.999999E+09,8.999999E+09,8.999999E+09]];
	LOCAL CONST Robtarget Tr_meulage_bavure_P149 :=[[-43.09426953125,-179.271671875,53],[0.708356088393271,-0.705687888858964,0.0108481326175781,-0.0108891493090295],[0,0,0,0],[8.999999E+09,8.999999E+09,8.999999E+09,8.999999E+09,8.999999E+09,8.999999E+09]];
	LOCAL CONST Robtarget Tr_meulage_bavure_P150 :=[[-32.41354296875,-179.63609375,53],[0.708269062189582,-0.705772218353488,0.0109467342656584,-0.0109854610464325],[0,0,0,0],[8.999999E+09,8.999999E+09,8.999999E+09,8.999999E+09,8.999999E+09,8.999999E+09]];
	LOCAL CONST Robtarget Tr_meulage_bavure_P151 :=[[-32.04992578125,-179.6458125,53],[0.70817698212268,-0.705858101646341,0.0111553430874596,-0.0111919905485173],[0,0,0,0],[8.999999E+09,8.999999E+09,8.999999E+09,8.999999E+09,8.999999E+09,8.999999E+09]];
	LOCAL CONST Robtarget Tr_meulage_bavure_P152 :=[[-22.3580625,-179.896703125,53],[0.708080546576137,-0.705946934636207,0.0114034601475795,-0.0114379252858691],[0,0,0,0],[8.999999E+09,8.999999E+09,8.999999E+09,8.999999E+09,8.999999E+09,8.999999E+09]];
	LOCAL CONST Robtarget Tr_meulage_bavure_P153 :=[[-20.4645078125,-179.95540625,53],[0.707983441610525,-0.706037438646439,0.0116154396583617,-0.0116474545045541],[0,0,0,0],[8.999999E+09,8.999999E+09,8.999999E+09,8.999999E+09,8.999999E+09,8.999999E+09]];
	LOCAL CONST Robtarget Tr_meulage_bavure_P154 :=[[-11.66943359375,-180.3486875,53],[0.707888033613021,-0.706129104800331,0.0117373768663898,-0.0117666140274349],[0,0,0,0],[8.999999E+09,8.999999E+09,8.999999E+09,8.999999E+09,8.999999E+09,8.999999E+09]];
	LOCAL CONST Robtarget Tr_meulage_bavure_P155 :=[[-3.51657104492188,-180.450984375,53],[0.707792002357478,-0.706224580974465,0.0117623936552691,-0.0117884995539129],[0,0,0,0],[8.999999E+09,8.999999E+09,8.999999E+09,8.999999E+09,8.999999E+09,8.999999E+09]];
	LOCAL CONST Robtarget Tr_meulage_bavure_P156 :=[[-2.82110595703125,-180.47071875,53],[0.707697713743958,-0.706320254596819,0.0117283177366155,-0.0117511901920515],[0,0,0,0],[8.999999E+09,8.999999E+09,8.999999E+09,8.999999E+09,8.999999E+09,8.999999E+09]];
	LOCAL CONST Robtarget Tr_meulage_bavure_P157 :=[[7.6112978515625,-180.9056875,53],[0.707608972089024,-0.706410818436823,0.0116797915771912,-0.0116996018413745],[0,0,0,0],[8.999999E+09,8.999999E+09,8.999999E+09,8.999999E+09,8.999999E+09,8.999999E+09]];
	LOCAL CONST Robtarget Tr_meulage_bavure_P158 :=[[8.231201171875,-180.9303125,53],[0.707522776602458,-0.706498601147194,0.0116373157870789,-0.0116541858179253],[0,0,0,0],[8.999999E+09,8.999999E+09,8.999999E+09,8.999999E+09,8.999999E+09,8.999999E+09]];
	LOCAL CONST Robtarget Tr_meulage_bavure_P159 :=[[21.526123046875,-181.295640625,53],[0.707442394133297,-0.706581374584586,0.0115692193042555,-0.0115833172190076],[0,0,0,0],[8.999999E+09,8.999999E+09,8.999999E+09,8.999999E+09,8.999999E+09,8.999999E+09]];
	LOCAL CONST Robtarget Tr_meulage_bavure_P160 :=[[24.029205078125,-181.37734375,53],[0.707370330366147,-0.706658631922224,0.0114133940211434,-0.0114248888142412],[0,0,0,0],[8.999999E+09,8.999999E+09,8.999999E+09,8.999999E+09,8.999999E+09,8.999999E+09]];
	LOCAL CONST Robtarget Tr_meulage_bavure_P161 :=[[44.3929453125,-182.19159375,53],[0.70730690457474,-0.706731852952089,0.0111092268469418,-0.0111182661719674],[0,0,0,0],[8.999999E+09,8.999999E+09,8.999999E+09,8.999999E+09,8.999999E+09,8.999999E+09]];
	LOCAL CONST Robtarget Tr_meulage_bavure_P162 :=[[50.17834375,-182.38825,53],[0.707254231258282,-0.706800215090522,0.0106010351103674,-0.0106078447310103],[0,0,0,0],[8.999999E+09,8.999999E+09,8.999999E+09,8.999999E+09,8.999999E+09,8.999999E+09]];
	LOCAL CONST Robtarget Tr_meulage_bavure_P163 :=[[59.13043359375,-182.66775,53],[0.707210562381894,-0.706866232924451,0.00982992993723704,-0.00983471830352806],[0,0,0,0],[8.999999E+09,8.999999E+09,8.999999E+09,8.999999E+09,8.999999E+09,8.999999E+09]];
	LOCAL CONST Robtarget Tr_meulage_bavure_P164 :=[[68.0419609375,-182.990734375,53],[0.707174550365539,-0.706932897509606,0.0086597475795898,-0.00866270776540324],[0,0,0,0],[8.999999E+09,8.999999E+09,8.999999E+09,8.999999E+09,8.999999E+09,8.999999E+09]];
	LOCAL CONST Robtarget Tr_meulage_bavure_P165 :=[[75.31784375,-183.20728125,53],[0.707146070447472,-0.707002086639753,0.00679947442107913,-0.00680085916128871],[0,0,0,0],[8.999999E+09,8.999999E+09,8.999999E+09,8.999999E+09,8.999999E+09,8.999999E+09]];
	LOCAL CONST Robtarget Tr_meulage_bavure_P166 :=[[88.5849609375,-183.414015625,53],[0.707118136819387,-0.707076111055957,0.00369541145818872,-0.00369563109859983],[0,0,0,0],[8.999999E+09,8.999999E+09,8.999999E+09,8.999999E+09,8.999999E+09,8.999999E+09]];
	LOCAL CONST Robtarget Tr_meulage_bavure_P167 :=[[89.8160390625,-183.434546875,53],[0.707071508967076,-0.707139265098928,-0.00140380554215764,0.00140367103338673],[0,0,0,0],[8.999999E+09,8.999999E+09,8.999999E+09,8.999999E+09,8.999999E+09,8.999999E+09]];
	LOCAL CONST Robtarget Tr_meulage_bavure_P168 :=[[90.956359375,-183.4825625,53],[0.706944846990352,-0.707143969616591,-0.00939252960320909,0.00938988478794944],[0,0,0,0],[8.999999E+09,8.999999E+09,8.999999E+09,8.999999E+09,8.999999E+09,8.999999E+09]];
	LOCAL CONST Robtarget Tr_meulage_bavure_P169 :=[[93.7432265625,-183.653796875,53],[0.706604125058735,-0.706968748895538,-0.021286918837089,0.0212759399670438],[0,0,0,0],[8.999999E+09,8.999999E+09,8.999999E+09,8.999999E+09,8.999999E+09,8.999999E+09]];
	LOCAL CONST Robtarget Tr_meulage_bavure_P170 :=[[96.872984375,-183.241671875,53],[0.705796422607367,-0.706368143047662,-0.0380644243071486,0.03803361571302],[0,0,0,0],[8.999999E+09,8.999999E+09,8.999999E+09,8.999999E+09,8.999999E+09,8.999999E+09]];
	LOCAL CONST Robtarget Tr_meulage_bavure_P171 :=[[97.8514375,-183.125109375,53],[0.704088287377531,-0.704922667898541,-0.0606317300667088,0.0605599634221864],[0,0,0,0],[8.999999E+09,8.999999E+09,8.999999E+09,8.999999E+09,8.999999E+09,8.999999E+09]];
	LOCAL CONST Robtarget Tr_meulage_bavure_P172 :=[[99.878296875,-182.617921875,53],[0.700822618529453,-0.701977617869819,-0.0897261173577185,0.0895784864308576],[0,0,0,0],[8.999999E+09,8.999999E+09,8.999999E+09,8.999999E+09,8.999999E+09,8.999999E+09]];
	LOCAL CONST Robtarget Tr_meulage_bavure_P173 :=[[100.4377421875,-182.4620625,53],[0.695101802315461,-0.696642538924553,-0.125683037602826,0.125405069424949],[0,0,0,0],[8.999999E+09,8.999999E+09,8.999999E+09,8.999999E+09,8.999999E+09,8.999999E+09]];
	LOCAL CONST Robtarget Tr_meulage_bavure_P174 :=[[101.19796875,-181.974828125,53],[0.685896865388169,-0.687891363712577,-0.168099055262532,0.167611662482593],[0,0,0,0],[8.999999E+09,8.999999E+09,8.999999E+09,8.999999E+09,8.999999E+09,8.999999E+09]];
	LOCAL CONST Robtarget Tr_meulage_bavure_P175 :=[[103.160640625,-180.730359375,53],[0.672350998213466,-0.674854481836622,-0.215475522754747,0.21467618088635],[0,0,0,0],[8.999999E+09,8.999999E+09,8.999999E+09,8.999999E+09,8.999999E+09,8.999999E+09]];
	LOCAL CONST Robtarget Tr_meulage_bavure_P176 :=[[103.68084375,-179.872359375,53],[0.654226739825638,-0.657276593968427,-0.265165855109161,0.263935448931378],[0,0,0,0],[8.999999E+09,8.999999E+09,8.999999E+09,8.999999E+09,8.999999E+09,8.999999E+09]];
	LOCAL CONST Robtarget Tr_meulage_bavure_P177 :=[[105.1572578125,-176.63778125,53],[0.632290831930907,-0.635915993365545,-0.31379821525036,0.312009348167204],[0,0,0,0],[8.999999E+09,8.999999E+09,8.999999E+09,8.999999E+09,8.999999E+09,8.999999E+09]];
	LOCAL CONST Robtarget Tr_meulage_bavure_P178 :=[[105.32546875,-175.589234375,53],[0.608325911247527,-0.61254275437573,-0.358113532767952,0.355648221442364],[0,0,0,0],[8.999999E+09,8.999999E+09,8.999999E+09,8.999999E+09,8.999999E+09,8.999999E+09]];
	LOCAL CONST Robtarget Tr_meulage_bavure_P179 :=[[105.3056015625,-174.6634375,53],[0.584574004971907,-0.589395426301721,-0.395878645041216,0.392640245728897],[0,0,0,0],[8.999999E+09,8.999999E+09,8.999999E+09,8.999999E+09,8.999999E+09,8.999999E+09]];
	LOCAL CONST Robtarget Tr_meulage_bavure_P180 :=[[105.289796875,-167.65553125,53],[0.563052544674233,-0.568494914745933,-0.426172606848259,0.422092730352045],[0,0,0,0],[8.999999E+09,8.999999E+09,8.999999E+09,8.999999E+09,8.999999E+09,8.999999E+09]];
	LOCAL CONST Robtarget Tr_meulage_bavure_P181 :=[[105.25396875,-167.26815625,53],[0.545091431331501,-0.551184665143304,-0.449169692822668,0.444204213678156],[0,0,0,0],[8.999999E+09,8.999999E+09,8.999999E+09,8.999999E+09,8.999999E+09,8.999999E+09]];
	LOCAL CONST Robtarget Tr_meulage_bavure_P182 :=[[105.3791484375,-166.074546875,53],[0.531190230867025,-0.537967550922998,-0.465757010607856,0.459889399589707],[0,0,0,0],[8.999999E+09,8.999999E+09,8.999999E+09,8.999999E+09,8.999999E+09,8.999999E+09]];
	LOCAL CONST Robtarget Tr_meulage_bavure_P183 :=[[105.73690625,-160.0610625,53],[0.521155399650476,-0.528653990955751,-0.477145057214007,0.470377084516191],[0,0,0,0],[8.999999E+09,8.999999E+09,8.999999E+09,8.999999E+09,8.999999E+09,8.999999E+09]];
	LOCAL CONST Robtarget Tr_meulage_bavure_P184 :=[[105.953890625,-155.90471875,53],[0.514347222299957,-0.522602100240278,-0.484610435879223,0.476955663740057],[0,0,0,0],[8.999999E+09,8.999999E+09,8.999999E+09,8.999999E+09,8.999999E+09,8.999999E+09]];
	LOCAL CONST Robtarget Tr_meulage_bavure_P185 :=[[106.027953125,-154.511640625,53],[0.509966193274231,-0.518996299070313,-0.489303687513003,0.480790208568027],[0,0,0,0],[8.999999E+09,8.999999E+09,8.999999E+09,8.999999E+09,8.999999E+09,8.999999E+09]];
	LOCAL CONST Robtarget Tr_meulage_bavure_P186 :=[[106.033046875,-152.9475,53],[0.507246948915943,-0.517053423687867,-0.492167356513265,0.482832872794373],[0,0,0,0],[8.999999E+09,8.999999E+09,8.999999E+09,8.999999E+09,8.999999E+09,8.999999E+09]];
	LOCAL CONST Robtarget Tr_meulage_bavure_P187 :=[[106.081484375,-148.023859375,53],[0.505541954289589,-0.516106282524252,-0.49393691376197,0.483826376725536],[0,0,0,0],[8.999999E+09,8.999999E+09,8.999999E+09,8.999999E+09,8.999999E+09,8.999999E+09]];
	LOCAL CONST Robtarget Tr_meulage_bavure_P188 :=[[106.092953125,-146.666484375,53],[0.50440543612726,-0.515695287457009,-0.495100397752721,0.484261419736282],[0,0,0,0],[8.999999E+09,8.999999E+09,8.999999E+09,8.999999E+09,8.999999E+09,8.999999E+09]];
	LOCAL CONST Robtarget Tr_meulage_bavure_P189 :=[[106.1058671875,-145.102765625,53],[0.50352150145886,-0.515487324406677,-0.495997791475224,0.48448437208682],[0,0,0,0],[8.999999E+09,8.999999E+09,8.999999E+09,8.999999E+09,8.999999E+09,8.999999E+09]];
	LOCAL CONST Robtarget Tr_meulage_bavure_P190 :=[[106.1837734375,-143.357328125,53],[0.502662443425527,-0.515229852000423,-0.496873041296991,0.484753389270646],[0,0,0,0],[8.999999E+09,8.999999E+09,8.999999E+09,8.999999E+09,8.999999E+09,8.999999E+09]];
	LOCAL CONST Robtarget Tr_meulage_bavure_P191 :=[[106.4053671875,-137.835171875,53],[0.501694834728123,-0.514780560772795,-0.497867923235427,0.485212116574608],[0,0,0,0],[8.999999E+09,8.999999E+09,8.999999E+09,8.999999E+09,8.999999E+09,8.999999E+09]];
	LOCAL CONST Robtarget Tr_meulage_bavure_P192 :=[[106.56246875,-133.68015625,53],[0.500544845487442,-0.514055920146679,-0.49905990762567,0.485942977332486],[0,0,0,0],[8.999999E+09,8.999999E+09,8.999999E+09,8.999999E+09,8.999999E+09,8.999999E+09]];
	LOCAL CONST Robtarget Tr_meulage_bavure_P193 :=[[106.760953125,-128.121875,53],[0.499216675580945,-0.513049431954776,-0.500442671433697,0.486949816512026],[0,0,0,0],[8.999999E+09,8.999999E+09,8.999999E+09,8.999999E+09,8.999999E+09,8.999999E+09]];
	LOCAL CONST Robtarget Tr_meulage_bavure_P194 :=[[106.880859375,-123.697375,53],[0.497823234704309,-0.511869640319347,-0.501894752006124,0.488122071019733],[0,0,0,0],[8.999999E+09,8.999999E+09,8.999999E+09,8.999999E+09,8.999999E+09,8.999999E+09]];
	LOCAL CONST Robtarget Tr_meulage_bavure_P195 :=[[107.012265625,-120.0938125,53],[0.496581295219048,-0.51073412730643,-0.50318776639745,0.489244049724734],[0,0,0,0],[8.999999E+09,8.999999E+09,8.999999E+09,8.999999E+09,8.999999E+09,8.999999E+09]];
	LOCAL CONST Robtarget Tr_meulage_bavure_P196 :=[[107.065796875,-114.540515625,53],[0.495780568760462,-0.509940071042652,-0.504021125966238,0.490025974989381],[0,0,0,0],[8.999999E+09,8.999999E+09,8.999999E+09,8.999999E+09,8.999999E+09,8.999999E+09]];
	LOCAL CONST Robtarget Tr_meulage_bavure_P197 :=[[107.081546875,-111.7237421875,53],[0.495715203763333,-0.509784853618069,-0.504092603710144,0.490180055351306],[0,0,0,0],[8.999999E+09,8.999999E+09,8.999999E+09,8.999999E+09,8.999999E+09,8.999999E+09]];
	LOCAL CONST Robtarget Tr_meulage_bavure_P198 :=[[106.9865703125,-109.0600703125,53],[0.496565590884743,-0.510449226405001,-0.503215550165894,0.489528662371326],[0,0,0,0],[8.999999E+09,8.999999E+09,8.999999E+09,8.999999E+09,8.999999E+09,8.999999E+09]];
	LOCAL CONST Robtarget Tr_meulage_bavure_P199 :=[[106.828921875,-105.84303125,53],[0.498314014465894,-0.511917806725417,-0.501401763270371,0.48807742616688],[0,0,0,0],[8.999999E+09,8.999999E+09,8.999999E+09,8.999999E+09,8.999999E+09,8.999999E+09]];
	LOCAL CONST Robtarget Tr_meulage_bavure_P200 :=[[106.966796875,-102.8728515625,53],[0.500725596609138,-0.513948210478946,-0.498885175244291,0.48605009594422],[0,0,0,0],[8.999999E+09,8.999999E+09,8.999999E+09,8.999999E+09,8.999999E+09,8.999999E+09]];
	LOCAL CONST Robtarget Tr_meulage_bavure_P201 :=[[107.057828125,-99.0538359375,53],[0.503418724466123,-0.51614684304426,-0.496058822951685,0.483826072513805],[0,0,0,0],[8.999999E+09,8.999999E+09,8.999999E+09,8.999999E+09,8.999999E+09,8.999999E+09]];
	LOCAL CONST Robtarget Tr_meulage_bavure_P202 :=[[107.042875,-97.8974453125,53],[0.505979086455442,-0.518091005455814,-0.493363245688687,0.481829411658342],[0,0,0,0],[8.999999E+09,8.999999E+09,8.999999E+09,8.999999E+09,8.999999E+09,8.999999E+09]];
	LOCAL CONST Robtarget Tr_meulage_bavure_P203 :=[[107.095765625,-97.8218046875,53],[0.508079225708441,-0.519458543120174,-0.491157630881211,0.480398276443759],[0,0,0,0],[8.999999E+09,8.999999E+09,8.999999E+09,8.999999E+09,8.999999E+09,8.999999E+09]];
	LOCAL CONST Robtarget Tr_meulage_bavure_P204 :=[[107.1916484375,-96.6414609375,53],[0.509568317046976,-0.520107739881023,-0.48961468033523,0.479693166490829],[0,0,0,0],[8.999999E+09,8.999999E+09,8.999999E+09,8.999999E+09,8.999999E+09,8.999999E+09]];
	LOCAL CONST Robtarget Tr_meulage_bavure_P205 :=[[107.8136328125,-87.4205,53],[0.510477734865384,-0.520080531399533,-0.488705928825227,0.479682434738816],[0,0,0,0],[8.999999E+09,8.999999E+09,8.999999E+09,8.999999E+09,8.999999E+09,8.999999E+09]];
	LOCAL CONST Robtarget Tr_meulage_bavure_P206 :=[[108.06103125,-84.4635,53],[0.510968008853237,-0.519560601704158,-0.48825633172106,0.480181454889363],[0,0,0,0],[8.999999E+09,8.999999E+09,8.999999E+09,8.999999E+09,8.999999E+09,8.999999E+09]];
	LOCAL CONST Robtarget Tr_meulage_bavure_P207 :=[[108.224703125,-81.1767578125,53],[0.511239307034492,-0.518772190254464,-0.488045510885938,0.480958797471843],[0,0,0,0],[8.999999E+09,8.999999E+09,8.999999E+09,8.999999E+09,8.999999E+09,8.999999E+09]];
	LOCAL CONST Robtarget Tr_meulage_bavure_P208 :=[[108.4034765625,-77.16671875,53],[0.51145407403314,-0.517898103609468,-0.487895056092449,0.48182434420976],[0,0,0,0],[8.999999E+09,8.999999E+09,8.999999E+09,8.999999E+09,8.999999E+09,8.999999E+09]];
	LOCAL CONST Robtarget Tr_meulage_bavure_P209 :=[[108.7163125,-70.2783203125,53],[0.511675222884651,-0.517021349411347,-0.487735353034594,0.482692050834725],[0,0,0,0],[8.999999E+09,8.999999E+09,8.999999E+09,8.999999E+09,8.999999E+09,8.999999E+09]];
	LOCAL CONST Robtarget Tr_meulage_bavure_P210 :=[[108.9066171875,-67.4650078125,53],[0.51184612804909,-0.516108067666907,-0.487625298374262,0.48359856500583],[0,0,0,0],[8.999999E+09,8.999999E+09,8.999999E+09,8.999999E+09,8.999999E+09,8.999999E+09]];
	LOCAL CONST Robtarget Tr_meulage_bavure_P211 :=[[109.014921875,-58.42633203125,53],[0.511847747431125,-0.515054460176656,-0.487690042636788,0.484653699887605],[0,0,0,0],[8.999999E+09,8.999999E+09,8.999999E+09,8.999999E+09,8.999999E+09,8.999999E+09]];
	LOCAL CONST Robtarget Tr_meulage_bavure_P212 :=[[108.9866328125,-54.887296875,53],[0.511565898950026,-0.513770105807865,-0.488047138556138,0.485953289891933],[0,0,0,0],[8.999999E+09,8.999999E+09,8.999999E+09,8.999999E+09,8.999999E+09,8.999999E+09]];
	LOCAL CONST Robtarget Tr_meulage_bavure_P213 :=[[109.087375,-53.8453671875,53],[0.510981186259104,-0.512247652157527,-0.488712651948733,0.487504373286617],[0,0,0,0],[8.999999E+09,8.999999E+09,8.999999E+09,8.999999E+09,8.999999E+09,8.999999E+09]];
	LOCAL CONST Robtarget Tr_meulage_bavure_P214 :=[[109.294765625,-51.1371171875,53],[0.510215998425109,-0.510628383380894,-0.489553488991823,0.489158124181556],[0,0,0,0],[8.999999E+09,8.999999E+09,8.999999E+09,8.999999E+09,8.999999E+09,8.999999E+09]];
	LOCAL CONST Robtarget Tr_meulage_bavure_P215 :=[[109.5556328125,-47.5888359375,53],[0.50952776396088,-0.50917874241483,-0.490300311900021,0.490636393041343],[0,0,0,0],[8.999999E+09,8.999999E+09,8.999999E+09,8.999999E+09,8.999999E+09,8.999999E+09]];
	LOCAL CONST Robtarget Tr_meulage_bavure_P216 :=[[109.62496875,-45.6123359375,53],[0.509203916823529,-0.508188384402423,-0.490659143437158,0.491639646500916],[0,0,0,0],[8.999999E+09,8.999999E+09,8.999999E+09,8.999999E+09,8.999999E+09,8.999999E+09]];
	LOCAL CONST Robtarget Tr_meulage_bavure_P217 :=[[109.6987578125,-42.92916796875,53],[0.509428913912466,-0.507840507701181,-0.490445289014885,0.491979287054728],[0,0,0,0],[8.999999E+09,8.999999E+09,8.999999E+09,8.999999E+09,8.999999E+09,8.999999E+09]];
	LOCAL CONST Robtarget Tr_meulage_bavure_P218 :=[[109.70825,-36.91064453125,53],[0.510175284247897,-0.508103863968052,-0.48968993829087,0.491686289314636],[0,0,0,0],[8.999999E+09,8.999999E+09,8.999999E+09,8.999999E+09,8.999999E+09,8.999999E+09]];
	LOCAL CONST Robtarget Tr_meulage_bavure_P219 :=[[109.7842734375,-34.00079296875,53],[0.511201090606738,-0.508725127468614,-0.488642168203519,0.491020387660114],[0,0,0,0],[8.999999E+09,8.999999E+09,8.999999E+09,8.999999E+09,8.999999E+09,8.999999E+09]];
	LOCAL CONST Robtarget Tr_meulage_bavure_P220 :=[[110.0485546875,-29.598052734375,53],[0.512140136511317,-0.509329247666655,-0.487680150419573,0.490371562116148],[0,0,0,0],[8.999999E+09,8.999999E+09,8.999999E+09,8.999999E+09,8.999999E+09,8.999999E+09]];
	LOCAL CONST Robtarget Tr_meulage_bavure_P221 :=[[110.2209140625,-27.414734375,53],[0.512655085915286,-0.509562654238284,-0.487155735803375,0.490112184468718],[0,0,0,0],[8.999999E+09,8.999999E+09,8.999999E+09,8.999999E+09,8.999999E+09,8.999999E+09]];
	LOCAL CONST Robtarget Tr_meulage_bavure_P222 :=[[110.2939765625,-21.9833984375,53],[0.512563771947017,-0.509227117191994,-0.487259972969843,0.490452690425087],[0,0,0,0],[8.999999E+09,8.999999E+09,8.999999E+09,8.999999E+09,8.999999E+09,8.999999E+09]];
	LOCAL CONST Robtarget Tr_meulage_bavure_P223 :=[[110.3570859375,-20.797423828125,53],[0.511880469125749,-0.5083210923637,-0.487976243175082,0.491393160801523],[0,0,0,0],[8.999999E+09,8.999999E+09,8.999999E+09,8.999999E+09,8.999999E+09,8.999999E+09]];
	LOCAL CONST Robtarget Tr_meulage_bavure_P224 :=[[110.2679140625,-15.5063173828125,53],[0.510778979622935,-0.506992556355121,-0.489119915363794,0.492772858597516],[0,0,0,0],[8.999999E+09,8.999999E+09,8.999999E+09,8.999999E+09,8.999999E+09,8.999999E+09]];
	LOCAL CONST Robtarget Tr_meulage_bavure_P225 :=[[110.25375,-15.0229794921875,53],[0.50950834135012,-0.50547180103083,-0.490429767084217,0.494346186406874],[0,0,0,0],[8.999999E+09,8.999999E+09,8.999999E+09,8.999999E+09,8.999999E+09,8.999999E+09]];
	LOCAL CONST Robtarget Tr_meulage_bavure_P226 :=[[110.3193984375,-11.937744140625,53],[0.508317673557579,-0.50399418575265,-0.491649299406541,0.495866887248575],[0,0,0,0],[8.999999E+09,8.999999E+09,8.999999E+09,8.999999E+09,8.999999E+09,8.999999E+09]];
	LOCAL CONST Robtarget Tr_meulage_bavure_P227 :=[[110.4932265625,-4.91046142578125,53],[0.507393327167469,-0.50273101872737,-0.492591151372972,0.497159423067004],[0,0,0,0],[8.999999E+09,8.999999E+09,8.999999E+09,8.999999E+09,8.999999E+09,8.999999E+09]];
	LOCAL CONST Robtarget Tr_meulage_bavure_P228 :=[[110.5030234375,-4.3906552734375,53],[0.506831457341342,-0.501774953228592,-0.493161905676576,0.498131614085217],[0,0,0,0],[8.999999E+09,8.999999E+09,8.999999E+09,8.999999E+09,8.999999E+09,8.999999E+09]];
	LOCAL CONST Robtarget Tr_meulage_bavure_P229 :=[[110.4938671875,-2.23825073242188,53],[0.506631796199839,-0.501129695433425,-0.493365448670057,0.49878230270602],[0,0,0,0],[8.999999E+09,8.999999E+09,8.999999E+09,8.999999E+09,8.999999E+09,8.999999E+09]];
	LOCAL CONST Robtarget Tr_meulage_bavure_P230 :=[[110.4480625,4.06185913085938,53],[0.50671212106992,-0.500717888626196,-0.493286714740822,0.499191986545011],[0,0,0,0],[8.999999E+09,8.999999E+09,8.999999E+09,8.999999E+09,8.999999E+09,8.999999E+09]];
	LOCAL CONST Robtarget Tr_meulage_bavure_P231 :=[[110.4958203125,7.893158203125,53],[0.506935608043394,-0.500417533167878,-0.493063958313153,0.499486250870247],[0,0,0,0],[8.999999E+09,8.999999E+09,8.999999E+09,8.999999E+09,8.999999E+09,8.999999E+09]];
	LOCAL CONST Robtarget Tr_meulage_bavure_P232 :=[[110.6371484375,10.3306884765625,53],[0.507146558612185,-0.500099350817883,-0.492853396131219,0.499798496717701],[0,0,0,0],[8.999999E+09,8.999999E+09,8.999999E+09,8.999999E+09,8.999999E+09,8.999999E+09]];
	LOCAL CONST Robtarget Tr_meulage_bavure_P233 :=[[110.663484375,11.1839599609375,53],[0.50721734363503,-0.499662822964949,-0.49278249382021,0.500232989162907],[0,0,0,0],[8.999999E+09,8.999999E+09,8.999999E+09,8.999999E+09,8.999999E+09,8.999999E+09]];
	LOCAL CONST Robtarget Tr_meulage_bavure_P234 :=[[110.749265625,18.1617734375,53],[0.507076664215007,-0.499056218683782,-0.492921738426069,0.500843595335557],[0,0,0,0],[8.999999E+09,8.999999E+09,8.999999E+09,8.999999E+09,8.999999E+09,8.999999E+09]];
	LOCAL CONST Robtarget Tr_meulage_bavure_P235 :=[[110.7666640625,20.653044921875,53],[0.506717582386548,-0.498305967361979,-0.493276980066313,0.501603703662994],[0,0,0,0],[8.999999E+09,8.999999E+09,8.999999E+09,8.999999E+09,8.999999E+09,8.999999E+09]];
	LOCAL CONST Robtarget Tr_meulage_bavure_P236 :=[[110.771546875,21.85174609375,53],[0.506220688876302,-0.49751753865662,-0.493767367825028,0.502404915734116],[0,0,0,0],[8.999999E+09,8.999999E+09,8.999999E+09,8.999999E+09,8.999999E+09,8.999999E+09]];
	LOCAL CONST Robtarget Tr_meulage_bavure_P237 :=[[110.766296875,22.30224609375,53],[0.505753239163661,-0.49687382769854,-0.494227627834475,0.503059750237259],[0,0,0,0],[8.999999E+09,8.999999E+09,8.999999E+09,8.999999E+09,8.999999E+09,8.999999E+09]];
	LOCAL CONST Robtarget Tr_meulage_bavure_P238 :=[[110.8980078125,28.839203125,53],[0.505534362296236,-0.496606498588436,-0.494443021326631,0.503331990597522],[0,0,0,0],[8.999999E+09,8.999999E+09,8.999999E+09,8.999999E+09,8.999999E+09,8.999999E+09]];
	LOCAL CONST Robtarget Tr_meulage_bavure_P239 :=[[110.89328125,29.109435546875,53],[0.505750091725516,-0.496905817674325,-0.494231168536568,0.50302783732913],[0,0,0,0],[8.999999E+09,8.999999E+09,8.999999E+09,8.999999E+09,8.999999E+09,8.999999E+09]];
	LOCAL CONST Robtarget Tr_meulage_bavure_P240 :=[[110.663390625,34.54339453125,53],[0.506456815029548,-0.497830928611948,-0.493534133942572,0.502085570058578],[0,0,0,0],[8.999999E+09,8.999999E+09,8.999999E+09,8.999999E+09,8.999999E+09,8.999999E+09]];
	LOCAL CONST Robtarget Tr_meulage_bavure_P241 :=[[110.643828125,41.30282421875,53],[0.507534537483405,-0.499256338346008,-0.492464518902207,0.500630102476129],[0,0,0,0],[8.999999E+09,8.999999E+09,8.999999E+09,8.999999E+09,8.999999E+09,8.999999E+09]];
	LOCAL CONST Robtarget Tr_meulage_bavure_P242 :=[[110.6267109375,42.9426875,53],[0.508712947336869,-0.500899950028213,-0.491285147947154,0.4989481743429],[0,0,0,0],[8.999999E+09,8.999999E+09,8.999999E+09,8.999999E+09,8.999999E+09,8.999999E+09]];
	LOCAL CONST Robtarget Tr_meulage_bavure_P243 :=[[110.9578828125,49.11047265625,53],[0.509695660000462,-0.502448962845884,-0.490291405170302,0.497362756876628],[0,0,0,0],[8.999999E+09,8.999999E+09,8.999999E+09,8.999999E+09,8.999999E+09,8.999999E+09]];
	LOCAL CONST Robtarget Tr_meulage_bavure_P244 :=[[111.0017421875,50.8075859375,53],[0.510290147660942,-0.503678565845908,-0.48968120312318,0.496109047302524],[0,0,0,0],[8.999999E+09,8.999999E+09,8.999999E+09,8.999999E+09,8.999999E+09,8.999999E+09]];
	LOCAL CONST Robtarget Tr_meulage_bavure_P245 :=[[111.1690703125,52.5979296875,53],[0.510476952376042,-0.504532407506002,-0.489479938513905,0.495247130896776],[0,0,0,0],[8.999999E+09,8.999999E+09,8.999999E+09,8.999999E+09,8.999999E+09,8.999999E+09]];
	LOCAL CONST Robtarget Tr_meulage_bavure_P246 :=[[111.279234375,53.5479140625,53],[0.510389207439198,-0.505103875754295,-0.489556453097859,0.494679098868975],[0,0,0,0],[8.999999E+09,8.999999E+09,8.999999E+09,8.999999E+09,8.999999E+09,8.999999E+09]];
	LOCAL CONST Robtarget Tr_meulage_bavure_P247 :=[[111.695890625,62.11969140625,53],[0.510216693804022,-0.505538631105449,-0.489719602035641,0.494251281440701],[0,0,0,0],[8.999999E+09,8.999999E+09,8.999999E+09,8.999999E+09,8.999999E+09,8.999999E+09]];
	LOCAL CONST Robtarget Tr_meulage_bavure_P248 :=[[111.828734375,70.5426015625,53],[0.510103392542383,-0.505943274251718,-0.489823494052276,0.493851067459232],[0,0,0,0],[8.999999E+09,8.999999E+09,8.999999E+09,8.999999E+09,8.999999E+09,8.999999E+09]];
	LOCAL CONST Robtarget Tr_meulage_bavure_P249 :=[[111.846859375,73.557921875,53],[0.510091835422997,-0.506326005729112,-0.489825504862397,0.493468611102569],[0,0,0,0],[8.999999E+09,8.999999E+09,8.999999E+09,8.999999E+09,8.999999E+09,8.999999E+09]];
	LOCAL CONST Robtarget Tr_meulage_bavure_P250 :=[[112.0394296875,81.33084375,53],[0.510135782954795,-0.506615052278385,-0.489773930726223,0.493177623716905],[0,0,0,0],[8.999999E+09,8.999999E+09,8.999999E+09,8.999999E+09,8.999999E+09,8.999999E+09]];
	LOCAL CONST Robtarget Tr_meulage_bavure_P251 :=[[112.2966328125,84.0065,53],[0.510161243205321,-0.506723173429264,-0.489745526085951,0.493068404098024],[0,0,0,0],[8.999999E+09,8.999999E+09,8.999999E+09,8.999999E+09,8.999999E+09,8.999999E+09]];
	LOCAL CONST Robtarget Tr_meulage_bavure_degg1 :=[[122.29060027019,83.6658504168746,52.9323810962286],[0.510161243205321,-0.506723173429264,-0.489745526085951,0.493068404098024],[0,0,0,0],[8.999999E+09,8.999999E+09,8.999999E+09,8.999999E+09,8.999999E+09,8.999999E+09]];
	LOCAL CONST Robtarget Tr_meulage_bavure_degg2 :=[[312.175981966303,77.1935083374912,51.6476219245717],[0.510161243205321,-0.506723173429264,-0.489745526085951,0.493068404098024],[0,0,0,0],[8.999999E+09,8.999999E+09,8.999999E+09,8.999999E+09,8.999999E+09,8.999999E+09]];
	LOCAL PROC Tr_pick()
		!!Programme Tr_pick - 27/03/2023 14:35:34;
		 CONST Robtarget Ppick :=[[-11.2277583818242,-29.0750951308758,141.121643991496],[0.0366721531145584,-0.683950290457426,0.726066923664886,0.0607780859270309],[0,0,0,0],[8.999999E+09,8.999999E+09,8.999999E+09,8.999999E+09,8.999999E+09,8.999999E+09]];
		 VAR Pose Ref :=[[0,0,0],[1,0,0,0]];
		LocalisationPieceTable 101 \model:=0;
		MoveJ Reltool(Ppick,0,0,-200),V1000,Z0,Tool_Prehenseur \Wobj:=Wobj_vision;
		MoveL Reltool(Ppick,0,0,-100),V500,Z0,Tool_Prehenseur \Wobj:=Wobj_vision;
		MoveL Reltool(Ppick,0,0,-10),V200,Z0,Tool_Prehenseur \Wobj:=Wobj_vision;
		MoveL Ppick,V100,Fine,Tool_Prehenseur \Wobj:=Wobj_vision;
		Gripper_Close;
		MoveL Reltool(Ppick,0,0,-200),V500,Z0,Tool_Prehenseur \Wobj:=Wobj_vision;
		LocalisationPiecePrehenseur 101 \model:=0,Ref;
	ENDPROC
	LOCAL PROC Tr_Cut()
		!!Programme Tr_Cut - 27/03/2023 14:35:34;
		confJ \off;
		confL \off;
		Tool := ToolOffset(Tool_M2_D490_S180);
		MoveAbsJ [[0,-40,40,0,90,0],[8.999999E+09,8.999999E+09,8.999999E+09,8.999999E+09,8.999999E+09,8.999999E+09]] ,V1000,Z0,Tool_M2_D490_S180 \Wobj:=Wobj_Part_0;
		Movej Reltool(Coupe_0,-200,0,-40.81869921875),V1000,Z0,Tool_M2_D490_S180 \Wobj:=Wobj_Part_0;
		MoveL Reltool(Coupe_0,0,0,-40.81869921875),V500,Z0,Tool_M2_D490_S180 \Wobj:=Wobj_Part_0;
		MoveL Reltool(Coupe_0,0,0,-30.81869921875),vitesse_Tronconnage,Z0,Tool_M2_D490_S180 \Wobj:=Wobj_Part_0;
		MoveL Coupe_0,vitesse_Tronconnage,Fine,Tool_M2_D490_S180 \Wobj:=Wobj_Part_0;
		MoveL Reltool(Coupe_0,0,0,30.81869921875),vitesse_Tronconnage,Z0,Tool_M2_D490_S180 \Wobj:=Wobj_Part_0;
		MoveL Reltool(Coupe_0,-200,0,30.81869921875),V500,Z0,Tool_M2_D490_S180 \Wobj:=Wobj_Part_0;
	ENDPROC
	LOCAL PROC Tr_meulage_motif_1()
		!!Programme Tr_meulage_motif_1 - 27/03/2023 14:35:34;
		 CONST Speeddata vitesse_Meulage :=[50, 500, 0, 0];
		confJ \off;
		confL \off;
		Tool := ToolOffset(Tool_M1_D500_S0);
		MoveAbsJ [[0,-40,40,0,90,0],[8.999999E+09,8.999999E+09,8.999999E+09,8.999999E+09,8.999999E+09,8.999999E+09]] ,V1000,Z0,Tool_M1_D500_S0 \Wobj:=Wobj_Part_0;
		MoveJ Tr_meulage_motif_1_App1,V2000,Z100,Tool,\Wobj:=Wobj_Part_0;
		MoveJ Tr_meulage_motif_1_App2,V500,Z0,Tool,\Wobj:=Wobj_Part_0;
		MoveL Tr_meulage_motif_1_P0,[12.5,500,0,0],z0,Tool \wobj:=Wobj_Part_0;
		MoveL Tr_meulage_motif_1_P1,[12.5,500,0,0],z0,Tool \wobj:=Wobj_Part_0;
		MoveL Tr_meulage_motif_1_P2,[12.5,500,0,0],z0,Tool \wobj:=Wobj_Part_0;
		MoveL Tr_meulage_motif_1_P3,[12.5,500,0,0],z0,Tool \wobj:=Wobj_Part_0;
		MoveL Tr_meulage_motif_1_P4,[12.5,500,0,0],z0,Tool \wobj:=Wobj_Part_0;
		MoveL Tr_meulage_motif_1_P5,[12.5,500,0,0],z0,Tool \wobj:=Wobj_Part_0;
		MoveL Tr_meulage_motif_1_P6,[12.5,500,0,0],z0,Tool \wobj:=Wobj_Part_0;
		MoveL Tr_meulage_motif_1_P7,[12.5,500,0,0],z0,Tool \wobj:=Wobj_Part_0;
		MoveL Tr_meulage_motif_1_P8,[12.5,500,0,0],z0,Tool \wobj:=Wobj_Part_0;
		MoveL Tr_meulage_motif_1_P9,[12.5,500,0,0],z0,Tool \wobj:=Wobj_Part_0;
		MoveL Tr_meulage_motif_1_P10,[12.5,500,0,0],z0,Tool \wobj:=Wobj_Part_0;
		MoveL Tr_meulage_motif_1_P11,[12.5,500,0,0],z0,Tool \wobj:=Wobj_Part_0;
		MoveL Tr_meulage_motif_1_P12,[12.5,500,0,0],z0,Tool \wobj:=Wobj_Part_0;
		MoveL Tr_meulage_motif_1_P13,[12.5,500,0,0],z0,Tool \wobj:=Wobj_Part_0;
		MoveL Tr_meulage_motif_1_P14,[12.5,500,0,0],z0,Tool \wobj:=Wobj_Part_0;
		MoveL Tr_meulage_motif_1_P15,[12.5,500,0,0],z0,Tool \wobj:=Wobj_Part_0;
